(* CODESYS project library.library
   Company: SLAC
   Title: lcls-twincat-motion
   Placeholder: lcls-twincat-motion
   Version: 0.2.0

Project tree, tasks and I/O mapping:
  libraries: Tc2_EtherCAT, * (Beckhoff Automation GmbH); Tc2_MC2, * (Beckhoff Automation GmbH); Tc2_Standard, * (Beckhoff Automation GmbH); Tc2_System, * (Beckhoff Automation GmbH); Tc2_Utilities, * (Beckhoff Automation GmbH); Tc3_Module, * (Beckhoff Automation GmbH); TcUnit, * (www.tcunit.org)
  DUTs/
    data type DUT_MotionStage
    data type DUT_PositionState
    data type EL5042_Status
    data type ENUM_EpicsHomeCmd
    data type ENUM_EpicsMotorCmd
    data type ENUM_StageBrakeMode
    data type ENUM_StageEnableMode
    data type ST_RenishawAbsEnc
  POUs/
    Motion/
      Gantry/
        function block FB_GantryAutoCoupling [ST]
        function block FB_GantryDiffVirtualLimitSwitch [ST]
      function block FB_MotionStage [ST]
      function block FB_SetEnables [ST]
      function block FB_StatePTPMove [ST]
    MotorTesting/
      function block FB_MicroStepCountTest [ST]
  tc_mca_std_lib/
    DUTs/
      data type DUT_AxisStatus_v0_01
    GVLs/
      global variables GVL
    POUs/
      ChangeConfig/
        function block FB_ReadFloatParameter [ST]
        function block FB_ReadParameterInNc_v1_00 [ST]
        function block FB_WriteFloatParameter [ST]
        function block FB_WriteParameterInNc_v1_00 [ST]
      ErrorHandling/
        data type DUT_ErrorState
        data type DUT_TerminalError
        function block FB_ErrorList [ST]
        function block FB_TerminalError [ST]
        global variables GVL_ErrorSystem
        data type ST_ErrorSystem
      Hardware/
        EtherCAT_Terminals/
          Analog_Inputs/
            function block EL3174_0002 [ST]
            function block EL3214 [ST]
            function block EL3255 [ST]
            function block FB_CalculateFrequency_3702_v0_01 [ST]
          Digital_Inputs/
            function block EL1008 [ST]
            function block EL1018 [ST]
            function block EL1808 [ST]
            function block EL1809 [ST]
            function block EL1819 [ST]
            function block FB_EL1252ASM_v1_00 [ST]
          Digital_Outputs/
            External_Types/
              data type dutEL2521_Ctrl
              data type dutEL2521_Status
            function block EL2014 [ST]
            function block EL2252 [ST]
            function block EL2808 [ST]
            function block EL2819 [ST]
          Measuring_Terminals/
            function block EL5002 [ST]
            function block EL5021 [ST]
            function block EL5042 [ST]
            function block EL5101 [ST]
          Motion/
            function block EL7211_v1_00 [ST]
            function block EL9576_v1_00 [ST]
          System/
            function block EL9410 [ST]
            function block EL9505 [ST]
        Other/
          function block EK1200 [ST]
      Motion/
        Homing/
          function block FB_HomeDirect [ST]
          function block FB_HomeFinish [ST]
          function block FB_HomePrepare [ST]
          function block FB_HomeReadNcVelocities [ST]
          function block FB_HomeReadSoftLimEnable [ST]
          function block FB_HomeToSwitch [ST]
          function block FB_HomeVirtual [ST]
          function block FB_HomeWriteNcVelocities [ST]
          function block FB_HomeWriteSoftLimEnable [ST]
        function block FB_DriveVirtual [ST]
        function block FB_NcAxis [ST]
  UnitTests/
    program Interactive [ST]
  Version/
    global variables Global_Version
*)

// DUTs/DUT_MotionStage
TYPE DUT_MotionStage :
STRUCT
	// Hardware
	Axis: AXIS_REF;
	bLimitForwardEnable AT %I*: BOOL;
	bLimitBackwardEnable AT %I*: BOOL;
	bHome AT %I*: BOOL;

	bBrakeRelease AT %Q*: BOOL;
	
	// Psuedo-hardware
	bAllForwardEnable: BOOL:=FALSE; // Forward enable EPS summary
	bAllBackwardEnable: BOOL:=FALSE; // Forward enable EPS summary
	bHardwareEnable AT %I*: BOOL; // True when Emergency stop button is not activated
	
	bAllEnable: BOOL:=FALSE; // Enable EPS summary encapsulating emergency stop button and any additional motion preventive hardware

	bGantryForwardEnable: BOOL:=FALSE; // Forward virtual gantry limit switch
	bGantryBackwardEnable: BOOL:=FALSE; // Reverse virtual gantry limit switch
	
	// Settings
	bPowerSelf: BOOL:=TRUE;
	nEnableMode: INT:=ENUM_StageEnableMode.STAGE_ENABLE_MOTION;
	nBrakeMode: INT:=ENUM_StageBrakeMode.STAGE_BRAKE_DISABLED;
	nHomingMode: INT:=ENUM_EpicsHomeCmd.EPICS_MOTOR_HOME_NONE;
	
	bGantryAxis: BOOL:=FALSE; // Set true to activate gantry EPS
	nGantryTol: LINT:=0; // Set to gantry difference tolerance
	nEncRef: ULINT:=0; // Encoder count at which this axis is aligned with other axis
	
	// Commands
	bEnable: BOOL;
	bReset: BOOL;
	bExecute: BOOL;
	
	// Args
	nCommand: INT;
	nCmdData: INT;
	fPosition: LREAL;
	fVelocity: LREAL;
	fAcceleration: LREAL;
	fDeceleration: LREAL;
	fHomePosition: LREAL;
	
	// Info
	nMotionAxisID: UDINT:=0;
	
	// Returns
	bEnableDone: BOOL;
	bBusy: BOOL;
	bDone: BOOL;
	bError: BOOL;
	sErrorMessage: STRING;
	stAxisStatus: DUT_AxisStatus_v0_01;
END_STRUCT
END_TYPE

// DUTs/DUT_PositionState
TYPE DUT_PositionState :
// Include io: input on things that should never be mutable in EPICS.
// Omit io on things that may or may not need to be mutable, allow engineer to decide in their pragma.
// Currently: some installations would want position and delta to be mutable.
STRUCT
	{attribute 'pytmc' := '
		pv: NAME
		io: input
	'}
	sName: STRING;

	{attribute 'pytmc' := '
		pv: SETPOINT
	'}
	fPosition: LREAL;
	
	{attribute 'pytmc' := '
		pv: DELTA
	'}
	fDelta: LREAL;
	
	{attribute 'pytmc' := '
		pv: VELO
		io: input
	'}
	fVelocity: LREAL;
	
	{attribute 'pytmc' := '
		pv: ACCL
		io: input
	'}
	fAccel: LREAL;
	
	{attribute 'pytmc' := '
		pv: DCCL
		io: input
	'}
	fDecel: LREAL;
END_STRUCT
END_TYPE

// DUTs/EL5042_Status
TYPE EL5042_Status :
STRUCT
END_STRUCT
END_TYPE

// DUTs/ENUM_EpicsHomeCmd
{attribute 'qualified_only'}
{attribute 'strict'}
TYPE ENUM_EpicsHomeCmd :
(
	EPICS_MOTOR_HOME_LLS := 1, // Low limit switch
	EPICS_MOTOR_HOME_HLS := 2, // High limit switch
	EPICS_MOTOR_HOME_LHS := 3, // Home switch via low switch
	EPICS_MOTOR_HOME_HHS := 4, // Home switch via high switch
	EPICS_MOTOR_HOME_ABS := 15, // Set here to be fHomePosition
	EPICS_MOTOR_HOME_NONE := -1 // Do not home, ever
);
END_TYPE

// DUTs/ENUM_EpicsMotorCmd
{attribute 'qualified_only'}
{attribute 'strict'}
TYPE ENUM_EpicsMotorCmd :
(
	EPICS_MOTOR_JOG := 0,
	EPICS_MOTOR_MOVE_VEL := 1,
	EPICS_MOTOR_MOVE_REL := 2,
	EPICS_MOTOR_MOVE_ABS := 3,
	EPICS_MOTOR_MOVE_MOD := 4,
	EPICS_MOTOR_HOME := 10,
	EPICS_MOTOR_GEAR := 30
);
END_TYPE

// DUTs/ENUM_StageBrakeMode
{attribute 'qualified_only'}
{attribute 'strict'}
TYPE ENUM_StageBrakeMode :
(
	STAGE_BRAKE_DISABLED,
	STAGE_BRAKE_STANDSTILL
);
END_TYPE

// DUTs/ENUM_StageEnableMode
{attribute 'qualified_only'}
{attribute 'strict'}
TYPE ENUM_StageEnableMode :
(
	STAGE_ENABLE_ALWAYS, // Always set bEnable to TRUE
	STAGE_ENABLE_NEVER,  // Only change bEnable on errors
	STAGE_ENABLE_MOTION  // Enable before motion, disable after motion
);
END_TYPE

// DUTs/ST_RenishawAbsEnc
// Renishaw BiSS-C absolute encoder used with an EL5042 
TYPE ST_RenishawAbsEnc :
STRUCT
	Count AT %I*: ULINT; // Connect to encoder "Position" input
	Status: EL5042_Status; // Status struct placeholder
	Ref: ULINT; // Encoder zero position (useful for aligned position with gantries)
END_STRUCT
END_TYPE

// tc_mca_std_lib/DUTs/DUT_AxisStatus_v0_01
TYPE DUT_AxisStatus_v0_01 :
STRUCT
	bEnable: BOOL;
	bReset: BOOL;
	bExecute: BOOL;
	nCommand: UINT;
	nCmdData: UINT;
	fVelocity: LREAL;
	fPosition: LREAL;
	fAcceleration: LREAL;
	fDeceleration: LREAL;
	bJogFwd: BOOL;
	bJogBwd: BOOL;
	bLimitFwd: BOOL;
	bLimitBwd: BOOL;
	fOverride: LREAL := 100;
	bHomeSensor: BOOL;
	bEnabled: BOOL;
	bError: BOOL;
	nErrorId: UDINT;
	fActVelocity: LREAL;
	fActPosition: LREAL;
	fActDiff: LREAL;
	bHomed:BOOL;
	bBusy:BOOL;
END_STRUCT
END_TYPE

// tc_mca_std_lib/POUs/ErrorHandling/DUT_ErrorState
{attribute 'qualified_only'}
{attribute 'strict'}
TYPE DUT_ErrorState :
(
	None,
	Active,
	Inactive,
	Acknowledged
);
END_TYPE

// tc_mca_std_lib/POUs/ErrorHandling/DUT_TerminalError
TYPE DUT_TerminalError :
STRUCT
	//Error system related
	iTerminalID : INT;					//ID of the terminal
	Error_ID : ULINT := 0;				//ID for the Error entry
	ErrorState : DUT_ErrorState;		//State of the error
	
	//Error related
	nDateTimeOn : ULINT;				//Date and time when the error occured. Raw data
	sDateTimeOn : STRING(24);			//Date and time when the error occured. Readable format
	nDateTimeOff : ULINT;				//Date and time when the error disapeared. Raw data
	sDateTimeOff : STRING(24);			//Date and time when the error disapeared. Readable format
	bWcState : BOOL;					//WcState variable of the terminal
	uiInfoDataState : UINT;				//InfoData.State variable of the terminal
	sErrorMessage : STRING (128);		//Error message corresponding to WcState and InfoData.State
	ErrorType : INT; 					//Error types (priorities) need to be developed
END_STRUCT
END_TYPE

// tc_mca_std_lib/POUs/ErrorHandling/ST_ErrorSystem
TYPE ST_ErrorSystem :
STRUCT
	//Array of error data. Size = cSizeOfErrorData in the GVL
	aErrorData : ARRAY [0..GVL_ErrorSystem.cSizeOfErrorData - 1] OF DUT_TerminalError;
	lNextErrorID : ULINT := 1;					//ErrorID for the next error entry
	nNoErrors : UINT;							//Number of errors in the list
	nNoOverflows : INT := 0;					//Number of overflows. How many error entries have been lost
END_STRUCT
END_TYPE

// tc_mca_std_lib/POUs/Hardware/EtherCAT_Terminals/Digital_Outputs/External_Types/dutEL2521_Ctrl
TYPE dutEL2521_Ctrl :
STRUCT
	///The control word (CW) is located in the output process image, and is transmitted from the controller to the terminal.
	///CW.0 FREQ_SEL 0bin / 1bin  Rapid change of the base frequency (only if the ramp function is inactive):
	///0bin = Base frequency 1 (object 8001:02)
	///1bin = Base frequency 2 (object 8001:03) 
	FREQ_SEL: BOOL;
	///CW.1 RAMP_DIS 1bin Operation of the ramp function is cancelled, in spite of object 8000:06 being active; if travel distance control is active, it is interrupted by this bit 
	RAMP_DIS: BOOL;
	///CW.2 GO_COUNTER 1bin  If travel distance control is active (object 8000:0A), then a pre-set counter value is approached when the bit is set 
	GO_COUNTER: BOOL;
	///CW.5 CNT_CLR 1bin The contents of the counter is cleared or set (object 8000:0B) by this bit. 
	///Any overflow or underflow bits that might be set are also cleared by this bit. 
	///The process can be edge triggered or level triggered (object 8000:05). 
	CNT_CLR: BOOL;
END_STRUCT
END_TYPE

// tc_mca_std_lib/POUs/Hardware/EtherCAT_Terminals/Digital_Outputs/External_Types/dutEL2521_Status
TYPE dutEL2521_Status :
STRUCT
	///The status word (SW) is located in the input process image, and is transmitted from the terminal to the controller.
	///SW.0 SEL_ACK/END_COUNTER 1bin  Confirms the change of base frequency. At activated travel distance control: target counter value reached 
	SEL_ACK: BOOL;
	///SW.1 RAMP_ACTIVE 1bin Ramp is currently being followed 
	RAMP_ACTIVE: BOOL;
	///SW.2 UNDERFLOW 1bin This bit is set if the 16-bit counter underflows (0 -> 65535). It is reset when the counter drops below two thirds of its measuring range (43690 -> 43689) or immediately an overflow occurs. 
	UNDERFLOW: BOOL;
	///SW.3 OVERFLOW 1bin This bit is set if the 16-bit counter overflows (65535 -> 0). It is reset when the counter exceeds one third of its measuring range (21845 -> 21846) or immediately an underflow occurs 
	OVERFLOW: BOOL;
	///SW.4 INPUT_T 1bin Status of INPUT_T 
	INPUT_T: BOOL;
	///SW.5 INPUT_Z 1bin Status of INPUT_Z 
	INPUT_Z: BOOL;
	///SW.6 ERROR 1bin General error bit, included with overflow/underflow 
	ERROR: BOOL;
END_STRUCT
END_TYPE

// tc_mca_std_lib/GVLs/GVL
VAR_GLOBAL
	nHomingError:UDINT:=16#14D00;
END_VAR

// tc_mca_std_lib/POUs/ErrorHandling/GVL_ErrorSystem
{attribute 'qualified_only'}
VAR_GLOBAL CONSTANT
	cSizeOfErrorData : UINT := 128;
	
END_VAR

// Version/Global_Version
{attribute 'TcGenerated'}
// This function has been automatically generated from the project information.
VAR_GLOBAL CONSTANT
	{attribute 'const_non_replaced'}
	{attribute 'linkalways'
	stLibVersion_lcls-twincat-motion : ST_LibVersion := (iMajor := 0, iMinor := 2, iBuild := 0, iRevision := 0, sVersion := '0.2.0');
END_VAR

// POUs/Motion/Gantry/FB_GantryAutoCoupling
FUNCTION_BLOCK FB_GantryAutoCoupling
VAR_INPUT
	nGantryTol : LINT;
END_VAR
VAR_OUTPUT
	bGantryAlreadyCoupled : BOOL;
END_VAR
VAR_IN_OUT
	Master : DUT_MotionStage;
	MasterEnc : ST_RenishawAbsEnc;
	Slave : DUT_MotionStage;
	SlaveEnc : ST_RenishawAbsEnc;
	bExecuteCouple : BOOL;
	bExecuteDecouple : BOOL;
END_VAR
VAR
	gantry_diff_limit : FB_GantryDiffVirtualLimitSwitch;
	couple : MC_GEARIN;
	decouple : MC_GEAROUT;
	bInitComplete : BOOL;
	fbSetEnables : FB_SetEnables;
END_VAR

// Designate Master and SLave Axes
Master.bGantryAxis := TRUE;
Slave.bGantryAxis := TRUE;

Master.nGantryTol := nGantryTol;
Slave.nGantryTol := Master.nGantryTol;

// Activate Gantry Virtual Limit Switch
gantry_diff_limit(Penc:=MasterEnc, SEnc:=SlaveEnc, GantDiffTol:=Master.nGantryTol,
				  PLimFwd=>Master.bGantryForwardEnable, PLimBwd=>Master.bGantryBackwardEnable,
				  SLimFwd=>Slave.bGantryForwardEnable, SLimBwd=>Slave.bGantryBackwardEnable);

// Coupling Status Bit
bGantryAlreadyCoupled := Master.Axis.NcToPlc.CoupleState=1 AND Slave.Axis.NcToPlc.CoupleState=3;

fbSetEnables(stMotionStage:=Master);
fbSetEnables(stMotionStage:=Slave);

IF bGantryAlreadyCoupled THEN
	Master.bGantryForwardEnable := Master.bGantryForwardEnable AND Slave.bAllForwardEnable;
	Slave.bGantryForwardEnable := Master.bAllForwardEnable AND Slave.bGantryForwardEnable;
	
	Master.bGantryBackwardEnable := Master.bGantryBackwardEnable AND Slave.bAllBackwardEnable;
	Slave.bGantryBackwardEnable := Master.bAllBackwardEnable AND Slave.bGantryBackwardEnable;
END_IF


// Coupling states
// Auto-coupling at init and auto-reset of coupling boolean
bExecuteCouple S= NOT bInitComplete;

bExecuteCouple R= couple.Busy OR bGantryAlreadyCoupled;
couple(Master:=Master.Axis, Slave:=Slave.Axis, Execute:=bExecuteCouple);

bInitComplete S= bGantryAlreadyCoupled;

// Decoupling with auto-reset of coupling boolean
bExecuteDecouple R= decouple.Busy OR NOT bGantryAlreadyCoupled;
decouple(Slave:=Slave.Axis, Execute:=bExecuteDecouple);

END_FUNCTION_BLOCK

// POUs/Motion/Gantry/FB_GantryDiffVirtualLimitSwitch
FUNCTION_BLOCK FB_GantryDiffVirtualLimitSwitch
VAR_INPUT
	PEnc: ST_RenishawAbsEnc; // Primary axis encoder (usually the upstream one)
	SEnc: ST_RenishawAbsEnc; // Secondary axis encoder (couples to the primary)
	
	GantDiffTol: LINT;		// Gantry differenace tolerance in encoder counts
END_VAR
VAR_OUTPUT
	PLimFwd: BOOL; // Primary axis forward direction enable
	PLimBwd: BOOL; // Primary axis reverse direction enable
	SLimFwd: BOOL; // Secondary axis forward direction enable
	SLimBwd: BOOL; // Secondary axis reverse direction enable
END_VAR
VAR
	GantryDiff: LINT;
END_VAR

(* Gantry Difference Virtual Limit Switch
A. Wallace 2017-2-15

Determines which direction is disabled due to it increasing the gantry difference.
Refer to the ESD for actual conventions.

A positive gantry error refers to a CCW clocked assembly:
eg. for X
X1 upstream, X2 downstream. Primary axis is always upstream.
Gantry difference > 0 when
X2>X1
Therefore
X2 positive direction disabled
X1 negative direction disabled

Call before FB_MotionStage fb calls for the gantry axes.
*)

GantryDiff := ( ULINT_TO_LINT(PEnc.Count) - ULINT_TO_LINT(PEnc.Ref) ) - ( ULINT_TO_LINT(SEnc.Count) - ULINT_TO_LINT(SEnc.Ref) );

IF ABS(GantryDiff) > GantDiffTol THEN
	IF GantryDiff < 0  THEN
		PLimBwd := FALSE;
		SLimFwd := FALSE;
	ELSE	
		PLimBwd := TRUE;
		SLimFwd := TRUE;
	END_IF
	IF GantryDiff > 0 THEN
		PLimFwd := FALSE;
		SLimBwd := FALSE;
	ELSE
		PLimFwd := TRUE;
		SLimBwd := TRUE;
	END_IF
ELSE
	//If there is no fault, all directions are enabled
	PLimFwd := TRUE;
	PLimBwd := TRUE;
	SLimFwd := TRUE;
	SLimBwd := TRUE;
END_IF

END_FUNCTION_BLOCK

// POUs/Motion/FB_MotionStage
FUNCTION_BLOCK FB_MotionStage
VAR_IN_OUT
	stMotionStage: DUT_MotionStage;
END_VAR
VAR
	fbDriveVirtual: FB_DriveVirtual;
	bExecute: BOOL;
	bFwdHit: BOOL;
	bBwdHit: BOOL;
	fbExecFallingEdge: F_TRIG;
	fbSetEnables: FB_SetEnables;
END_VAR

// Start with an accurate status
stMotionStage.Axis.ReadStatus();

// Handle auto-enable timing
CASE stMotionStage.nEnableMode OF
	ENUM_StageEnableMode.STAGE_ENABLE_ALWAYS:
		stMotionStage.bEnable := TRUE;
		bExecute := stMotionStage.bExecute;
	ENUM_StageEnableMode.STAGE_ENABLE_NEVER:
		bExecute := stMotionStage.bExecute;
	ENUM_StageEnableMode.STAGE_ENABLE_MOTION:
		IF stMotionStage.bExecute THEN
			stMotionStage.bEnable := TRUE;
		END_IF
		bExecute := stMotionStage.bExecute AND stMotionStage.bEnableDone;
END_CASE

// Automatically fill the correct nCmdData for homing
IF stMotionStage.nCommand = ENUM_EpicsMotorCmd.EPICS_MOTOR_HOME THEN
	stMotionStage.nCmdData := stMotionStage.nHomingMode;
END_IF

fbSetEnables(stMotionStage:=stMotionStage);

// Handle standard commands using ESS's FB
fbDriveVirtual(En:=TRUE,
	bEnable:=stMotionStage.bAllEnable,
	bReset:=stMotionStage.bReset,
	bExecute:=bExecute,
	nCommand:=INT_TO_UINT(stMotionStage.nCommand),
	nCmdData:=INT_TO_UINT(stMotionStage.nCmdData),
	fVelocity:=stMotionStage.fVelocity,
	fPosition:=stMotionStage.fPosition,
	fAcceleration:=stMotionStage.fAcceleration,
	fDeceleration:=stMotionStage.fDeceleration,
	bLimitFwd:=stMotionStage.bAllForwardEnable,
	bLimitBwd:=stMotionStage.bAllBackwardEnable,
	bHomeSensor:=stMotionStage.bHome,
	fHomePosition:=stMotionStage.fHomePosition,
	bPowerSelf:=stMotionStage.bPowerSelf,
	nMotionAxisID=>stMotionStage.nMotionAxisID,
	bError=>stMotionStage.bError,
	sErrorMessage=>stMotionStage.sErrorMessage,
	Axis:=stMotionStage.Axis);

IF fbDriveVirtual.bBusy THEN
	stMotionStage.bBusy := TRUE;
	stMotionStage.bDone := FALSE;
END_IF

IF stMotionStage.bError THEN
	stMotionStage.bBusy := FALSE;
	stMotionStage.bDone := FALSE;
	stMotionStage.bEnable := FALSE;
END_IF

// Check the limits and cancel execution if appropriate. Without this block we have infinite error spam
bFwdHit := stMotionStage.Axis.Status.PositiveDirection AND NOT stMotionStage.bAllForwardEnable;
bBwdHit := stMotionStage.Axis.Status.NegativeDirection AND NOT stMotionStage.bAllBackwardEnable;
IF bFwdHit OR bBwdHit THEN
	stMotionStage.bExecute := FALSE;
END_IF

// Mark done if settled or if unexpected stop, then reset the FB if there is no error
fbExecFallingEdge(CLK:=stMotionStage.bExecute);
IF (stMotionStage.Axis.Status.InTargetPosition AND NOT fbDriveVirtual.bBusy) OR fbExecFallingEdge.Q THEN
	IF NOT stMotionStage.bDone THEN
		stMotionStage.bDone := TRUE;
		stMotionStage.bBusy := FALSE;
		IF NOT stMotionStage.Axis.Status.Error THEN
			bExecute := FALSE;
			stMotionStage.bExecute := FALSE;
		END_IF
	END_IF
END_IF
IF stMotionStage.nEnableMode = ENUM_StageEnableMode.STAGE_ENABLE_MOTION AND NOT bExecute THEN
	IF stMotionStage.Axis.Status.MotionState = MC_AXISSTATE_STANDSTILL THEN
		stMotionStage.bEnable := FALSE;
	END_IF
END_IF

// Get a definitive bEnabled reading
CASE stMotionStage.Axis.Status.MotionState OF
	// We are not enabled if there is an issue
	MC_AXISSTATE_UNDEFINED, MC_AXISSTATE_DISABLED, MC_AXISSTATE_ERRORSTOP:
		stMotionStage.bEnableDone := FALSE;
	ELSE
		stMotionStage.bEnableDone := TRUE;
END_CASE

// Handle the brake. TRUE means brake disabled.
CASE stMotionStage.nBrakeMode OF
	ENUM_StageBrakeMode.STAGE_BRAKE_DISABLED:
		stMotionStage.bBrakeRelease := stMotionStage.bEnableDone AND stMotionStage.bExecute;
	ENUM_StageBrakeMode.STAGE_BRAKE_STANDSTILL:
		IF stMotionStage.Axis.Status.MotionState = MC_AXISSTATE_STANDSTILL THEN
			stMotionStage.bBrakeRelease := FALSE;
		ELSE
			stMotionStage.bBrakeRelease := TRUE;
		END_IF
END_CASE
CASE stMotionStage.Axis.Status.MotionState OF
	MC_AXISSTATE_UNDEFINED, MC_AXISSTATE_ERRORSTOP:
		stMotionStage.bBrakeRelease := FALSE;
END_CASE

// Sync the epics status struct
stMotionStage.stAxisStatus := fbDriveVirtual.stAxisStatus;
stMotionStage.stAxisStatus.bEnabled := stMotionStage.bEnableDone;

// Reset everything when bReset is flagged
IF stMotionStage.bReset THEN
	stMotionStage.bEnable := FALSE;
	stMotionStage.bReset := FALSE;
	stMotionStage.bExecute := FALSE;
	bExecute := FALSE;
END_IF

// Ignore homing if we have the setting for it
// e.g. for pre-calibrated absolute encoders
IF stMotionStage.nHomingMode = ENUM_EpicsHomeCmd.EPICS_MOTOR_HOME_NONE THEN
	stMotionStage.stAxisStatus.bHomed := TRUE;
END_IF

END_FUNCTION_BLOCK

// tc_mca_std_lib/POUs/Motion/FB_DriveVirtual
///#########################################################
///Function block to run a virtual drive with Nc
///	Library:		
///	Tc2_MC2.lib
///
///	Global Variables:
///	
///	Data types:
///	
///	External functions:
///
///###########################################################
FUNCTION_BLOCK FB_DriveVirtual
VAR
	sVersion: STRING:='1.0.3';	
END_VAR
VAR_INPUT
	En: BOOL;
	bEnable: BOOL;
	bReset: BOOL;
	bExecute: BOOL;
	/////	nCommandLocal...
	/////	0 = Jog
	/////	1 = MoveVelocity
	/////	2 = MoveRelative
	/////	3 = MoveAbsolut
	/////	4 = MoveModulo
	/////	10 = Homing
	/////	20 = SuperInp >>>ToBe
	/////	30 = Gear
	nCommand: UINT;
	nCmdData: UINT;
	fVelocity: LREAL;
	fPosition: LREAL;
	fAcceleration: LREAL;
	fDeceleration: LREAL;
	bJogFwd: BOOL;
	bJogBwd: BOOL;
	bLimitFwd: BOOL;
	bLimitBwd: BOOL;	
	fOverride: LREAL := 100;
	bHomeSensor: BOOL;
	fHomePosition:LREAL;
	nHomeRevOffset: UINT;
	MasterAxis: AXIS_REF;
	bPowerSelf: BOOL;
END_VAR
VAR_OUTPUT
	EnO: BOOL;
	bEnabled: BOOL;
	bBusy: BOOL;
	bDone: BOOL;
	bError: BOOL;
	bHomed: BOOL;
	nErrorId: UDINT;
	nMotionAxisID:UDINT:=0;  //Axis id in Motion (NC)
	Status: ST_AxisStatus;
	fActVelocity: LREAL;
	fActPosition: LREAL;
	fActDiff: LREAL;
    sErrorMessage:STRING;
END_VAR
VAR_IN_OUT
	Axis: AXIS_REF;
END_VAR
VAR	
	nCommandLocal: UINT;
	nCmdDataLocal: UINT;
	bFirstScan: BOOL := TRUE;
	fbReset: MC_Reset;
	fbPower: MC_Power;
	fbHalt: MC_Halt;
	fbJog: MC_Jog;
	fbMoveVelocity: MC_MoveVelocity;
	fbMoveRelative: MC_MoveRelative;
	fbMoveAbsolute: MC_MoveAbsolute;
	fbMoveModulo: MC_MoveModulo;	
	fbHomeVirtual:FB_HomeVirtual;
	fbGearInDyn: MC_GearInDyn;
	fbGearOut: MC_GearOut;
	fbExecuteRiseEdge: R_TRIG;
	stAxisStatus: DUT_AxisStatus_v0_01;	
END_VAR

EnO:=En;

// Transfer nCommand and nCmdData to local copies at rising edge of bExecute (avoid issues if nCommand or nCmdData are changed during a command) 
fbExecuteRiseEdge(CLK:=bExecute);
IF fbExecuteRiseEdge.Q THEN
  nCmdDataLocal:=nCmdData;
  nCommandLocal:=nCommand;
END_IF

bHomed:=fbHomeVirtual.bHomed; //Add in DUT_AxisStatus later
bDone:=FALSE;

(*Reset*)
fbReset(
	Execute:=bReset AND Axis.Status.Error,
	Axis:=Axis,
	Done=> ,
	Busy=> ,
	Error=> ,
	ErrorID=> );

(*Power*)
IF bPowerSelf THEN
fbPower(
	Axis:=Axis,
	Enable:=bEnable,	
	Enable_Positive:=bEnable AND bLimitFwd,	
	Enable_Negative:=bEnable AND bLimitBwd,	
	Override:=fOverride,
	BufferMode:= ,
	Status=> ,
	Busy=> ,
	Active=> ,
	Error=> ,
	ErrorID=> );
END_IF

(*Halt*)
fbHalt(
	Execute:=NOT bExecute  AND (((fbMoveVelocity.Busy OR fbPower.Busy) AND (nCommandLocal=1)) OR (fbMoveRelative.Busy AND (nCommandLocal=2)) OR (fbMoveAbsolute.Busy AND (nCommandLocal=3)) OR (fbMoveModulo.Busy AND (nCommandLocal=4)) OR (fbHomeVirtual.bBusy AND (nCommandLocal=10))),
	Deceleration:=fDeceleration,
	Jerk:=0,
	BufferMode:= ,
	Options:= ,
	Axis:=Axis ,
	Done=> ,
	Busy=> ,
	Active=> ,
	CommandAborted=> ,
	Error=> ,
	ErrorID=> );

(*Jog (Command = 0)*)
fbJog(
	JogForward:=bJogFwd AND (nCommandLocal=0) ,
	JogBackwards:=bJogBwd AND (nCommandLocal=0) ,
	Mode:=UINT_TO_INT(nCmdDataLocal),
	Position:= ,
	Velocity:=fVelocity,
	Acceleration:=fAcceleration,
	Deceleration:=fDeceleration,
	Jerk:=0,
	Axis:=Axis,
	Done=> ,
	Busy=> ,
	Active=> ,
	CommandAborted=> ,
	Error=> ,
	ErrorID=> );

(*MoveVelocity (Command = 1)*)
fbMoveVelocity(
	Execute:=bExecute AND (nCommandLocal=1),
	Velocity:=ABS(fVelocity),
	Acceleration:=fAcceleration,
	Deceleration:=fDeceleration,
	Jerk:=0,
	Direction:=SEL(fVelocity<0, MC_Positive_Direction, MC_Negative_Direction),
	BufferMode:= ,
	Options:= ,
	Axis:=Axis,
	InVelocity=> ,
	Busy=> ,
	Active=> ,
	CommandAborted=> ,
	Error=> ,
	ErrorID=> );

(*MoveRelative (Command = 2)*)
fbMoveRelative(
	Execute:=bExecute AND (nCommandLocal=2), 
	Distance:=fPosition, 
	Velocity:=ABS(fVelocity), 
	Acceleration:=fAcceleration,
	Deceleration:=fDeceleration,
	Jerk:=0,
	BufferMode:= , 
	Options:= , 
	Axis:=Axis, 
	Done=> , 
	Busy=> , 
	Active=> , 
	CommandAborted=> , 
	Error=> , 
	ErrorID=> );
	
IF nCommandLocal=2 THEN
	bDone:=fbMoveRelative.Done;
END_IF
	
(*MoveAbsolute (Command = 3)*)
fbMoveAbsolute(
	Execute:=bExecute AND (nCommandLocal=3),
	Position:=fPosition,
	Velocity:=ABS(fVelocity),
	Acceleration:=fAcceleration,
	Deceleration:=fDeceleration,
	Jerk:=0,
	BufferMode:= ,
	Options:= ,
	Axis:=Axis,
	Done=> ,
	Busy=> ,
	Active=> ,
	CommandAborted=> ,
	Error=> ,
	ErrorID=> );

IF nCommandLocal=3 THEN
	bDone:=fbMoveAbsolute.Done;
END_IF

(*MoveModulo (Command = 4)*)
fbMoveModulo(
	Execute:=bExecute AND (nCommandLocal=4), 
	Position:=fPosition, 
	Velocity:=ABS(fVelocity), 
	Acceleration:=fAcceleration, 
	Deceleration:=fDeceleration, 
	Jerk:=0, 
	Direction:=UINT_TO_INT(nCmdDataLocal), 
	BufferMode:= , 
	Options:= , 
	Axis:=Axis, 
	Done=> , 
	Busy=> , 
	Active=> , 
	CommandAborted=> , 
	Error=> , 
	ErrorID=> );

IF nCommandLocal=4 THEN
	bDone:=fbMoveModulo.Done;
END_IF
	
(*Home (Command = 10)*)
fbHomeVirtual(	
	bExecute:= nCommandLocal=10 AND bExecute,
	fHomePosition:=fHomePosition,
	bHomeSensor:=bHomeSensor,
	bLimitBwd:=bLimitBwd,
	bLimitFwd:=bLimitFwd,
	nCmdData:=nCmdDataLocal,
	bReset:=bReset,
	nHomeRevOffset:=nHomeRevOffset,
	Axis:=Axis
	);
	
IF nCommandLocal=10 THEN
	bDone:=fbHomeVirtual.bDone;
END_IF
	
(*Gear (Command = 30)*)
fbGearInDyn(
	Enable:=bExecute  AND (nCommandLocal=30),
	GearRatio:=SEL(nCmdDataLocal>0, 1,fVelocity),
	Acceleration:=fAcceleration,
	Deceleration:=fDeceleration,
	Jerk:=0.0,
	BufferMode:= , 
	Options:= , 
	Master:=MasterAxis,
	Slave:=Axis,
	InGear=> , 
	Busy=> , 
	Active=> , 
	CommandAborted=> , 
	Error=> , 
	ErrorID=> );
	
fbGearOut(
	Execute:=NOT bExecute AND Axis.Status.NotMoving AND (nCommandLocal=30),
	Slave:=Axis,
	Error=>,
	Done=>,
	ErrorID=>);


IF nCommandLocal=30 THEN
	bDone:=Axis.Status.Coupled;
END_IF

(*Busy*)
bBusy:=Axis.Status.HasJob OR Axis.Status.HomingBusy OR fbHomeVirtual.bBusy;

(*Enabled*)
bEnabled:=fbPower.Status;

(*Error from functions and Nc*)
IF fbPower.Error AND fbPower.Active THEN
	bError:=fbPower.Enable;
	nErrorId:=fbPower.ErrorID;
ELSIF fbHalt.Error AND fbHalt.Active THEN
	bError:=fbHalt.Execute;
	nErrorId:=fbHalt.ErrorID;
ELSIF fbJog.Error AND nCommandLocal=0 (*fbJog.Active*) THEN
	bError:=fbJog.JogForward OR fbJog.JogBackwards;
	nErrorId:=fbJog.ErrorID;
ELSIF fbMoveVelocity.Error AND nCommandLocal=1(*fbMoveVelocity.Active*) THEN
	bError:=fbMoveVelocity.Execute;
	nErrorId:=fbMoveVelocity.ErrorID;
ELSIF fbMoveRelative.Error AND nCommandLocal=2 (*fbMoveRelative.Active*) THEN
	bError:=fbMoveRelative.Execute;
	nErrorId:=fbMoveRelative.ErrorID;
ELSIF fbMoveAbsolute.Error AND nCommandLocal=3 (*fbMoveAbsolute.Active*) THEN
	bError:=fbMoveAbsolute.Execute;
	nErrorId:=fbMoveAbsolute.ErrorID;
ELSIF fbMoveModulo.Error AND nCommandLocal=4 (*fbMoveModulo.Active*) THEN
	bError:=fbMoveModulo.Execute;
	nErrorId:=fbMoveModulo.ErrorID;
ELSIF fbHomeVirtual.bError AND nCommandLocal=10 (*fbHome.Active*) THEN
	bError:=fbHomeVirtual.bError;
	nErrorId:=fbHomeVirtual.nErrorID;
ELSIF fbGearInDyn.Error AND nCommandLocal=30 (*fbGearInDyn.Active*) THEN
	bError:=fbGearInDyn.Enable;
	nErrorId:=fbGearInDyn.ErrorID;
ELSIF fbGearOut.Error AND nCommandLocal=30 AND Axis.Status.Coupled THEN
	bError:=fbGearOut.Execute;
	nErrorId:=fbGearOut.ErrorID;
ELSIF Axis.Status.Error  THEN
	bError:=TRUE;
	nErrorId:=Axis.Status.ErrorID;
ELSIF fbHomeVirtual.bError THEN
	bError:=TRUE;
	nErrorId:=fbHomeVirtual.nErrorId;
ELSE
	bError:=FALSE;
	nErrorId:=0;
END_IF;

(*Converese nErrorID to string*)
sErrorMessage:=WORD_TO_HEXSTR(in:=TO_WORD(nErrorID) , iPrecision:= 4, bLoCase:=0 );

(*Status from Nc*)
Status:=Axis.Status;

(*Axis id in motion "motor"*)
nMotionAxisID:=axis.NcToPlc.AxisId;

(*Actual Velocity*)
fActVelocity:=Axis.NcToPlc.ActVelo;

(*Actual Position*)
IF Axis.Status.OpMode.Modulo THEN
	fActPosition:=Axis.NcToPlc.ModuloActPos;
ELSE
	fActPosition:=Axis.NcToPlc.ActPos;
END_IF

(*Actual Position*)
fActDiff:=Axis.NcToPlc.PosDiff;


//Status struct for EPICS communication
stAxisStatus.bEnable:=bEnable;
stAxisStatus.bEnabled:=bEnabled;
stAxisStatus.bError:=bError;
stAxisStatus.bExecute:=bExecute;
stAxisStatus.bHomeSensor:=bHomeSensor;
stAxisStatus.bJogBwd:=bJogBwd;
stAxisStatus.bJogFwd:=bJogFwd;
stAxisStatus.bLimitBwd:=bLimitBwd;
stAxisStatus.bLimitFwd:=bLimitFwd;
stAxisStatus.bReset:=bReset;
stAxisStatus.fAcceleration:=fAcceleration;
stAxisStatus.fActDiff:=fActDiff;
stAxisStatus.fActPosition:=fActPosition;
stAxisStatus.fActVelocity:=fActVelocity;
stAxisStatus.fDeceleration:=fDeceleration;
stAxisStatus.fOverride:=fOverride;
stAxisStatus.fPosition:=fPosition;
stAxisStatus.fVelocity:=fVelocity;
stAxisStatus.nCmdData:=nCmdData;  //Or nCmdDataLocal
stAxisStatus.nCommand:=nCommand;  //Or nCommandLocal
stAxisStatus.nErrorId:=nErrorId;
stAxisStatus.bBusy:=bBusy;
stAxisStatus.bHomed:=bHomed;

IF bFirstScan THEN
	bFirstScan:=FALSE;
END_IF

END_FUNCTION_BLOCK

// tc_mca_std_lib/POUs/Motion/Homing/FB_HomeVirtual
FUNCTION_BLOCK FB_HomeVirtual
VAR_INPUT
	En: BOOL;
	bReset: BOOL;
	bExecute: BOOL;
	nCmdData: UINT;
	bLimitFwd: BOOL;
	bLimitBwd: BOOL;	
	bHomeSensor: BOOL;	
	fHomePosition:LREAL;
	nHomeRevOffset: UINT;
END_VAR
VAR_IN_OUT
	Axis: AXIS_REF;
END_VAR
VAR_OUTPUT
	EnO: BOOL;	
	bBusy: BOOL;
	bDone: BOOL;
	bHomed:BOOL;
	bError: BOOL;
	nErrorId: UDINT;
END_VAR
VAR
	fbHomeToSwitch: FB_HomeToSwitch;
    fbHomeDirect: FB_HomeDirect; //Only used for direct homing (set of position)
    fbMoveVelocity:MC_MoveVelocity;
    fbHomePrepare:FB_HomePrepare;
	fbHomeFinish:FB_HomeFinish;    	    		
	fbExecuteRiseEdge: R_TRIG;
    nHomingState:INT:=0;
	bExecuteHomeToSwitch:BOOL:=FALSE;
	bExecuteMoveVelocity:BOOL:=FALSE;
	bExecutePrepare: BOOL:=FALSE;
	bExecuteFinish: BOOL:=FALSE;
	bExecuteHomeDirect: BOOL;
	nCmdDataLocal: UINT;  //Ensure that nCmdData is not changed during sequence
	bSequenceReady:BOOL:=TRUE;
	bRestoreNCDataNeeded: BOOL:=FALSE;
END_VAR

EnO:=En;

IF bReset THEN	
	bError:=FALSE;
	nErrorId:=0;
END_IF

// Reset when bExecute is low
IF NOT bExecute THEN
  nHomingState:=0;
  bSequenceReady:=TRUE;
  bExecuteHomeToSwitch:=FALSE;
  bExecuteHomeDirect:=FALSE;
  bExecuteMoveVelocity:=FALSE;
  bExecutePrepare:=FALSE;
  bExecuteFinish:=FALSE;
END_IF

//Reset at rinsing edge of bExecute
fbExecuteRiseEdge(CLK:=bExecute);
IF fbExecuteRiseEdge.Q THEN
  nCmdDataLocal:=nCmdData; //Ensure that nCmdData is not changed during sequence (nCmdData will only be read at a rising edge of bExecute)
  bSequenceReady:=FALSE;
  bExecutePrepare:=TRUE;  
  bRestoreNCDataNeeded:=FALSE;
  //Check if valid nCmdDataLocal
  CASE nCmdDataLocal OF  	
    1:
    2:
    3:
    4:
    15:
    ELSE //nCmdData not valid	
      bError:=TRUE;
      nErrorId:=16#4FFF;   
  END_CASE
END_IF

//############# Prepare for homing (Read from NC and reset homed flag)
fbHomePrepare(
  En:=En,
  bExecute:=bExecutePrepare AND NOT bError, // Not needed for sequence 15 (set position only, no movement))
  bReset:=bReset,
  Axis:=Axis,
);

//############# Homing Sequences:
CASE nCmdDataLocal OF  
	
   1: // Home to low limit switch
	   CASE nHomingState OF
		  0:
		    bHomed:=Axis.Status.Homed;
            // Wait for read of velocities from NC and reset of calibration flag
	        IF fbHomePrepare.bDone AND bExecute AND NOT bSequenceReady THEN
			  bRestoreNCDataNeeded:=TRUE;
			  IF bLimitBwd THEN
                nHomingState:=1;
              ELSE
				nHomingState:=2;  //Standing on limit switch go direct to state 2 
              END_IF                                          		  
	        END_IF
		  1: // wait for reach low limit then trigger fbHomeToSwitch
		    bHomed:=FALSE;
			bSequenceReady:=FALSE;
			fbMoveVelocity.Velocity:=ABS(fbHomePrepare.fVelocityToCam);
            fbMoveVelocity.Direction:=MC_Negative_Direction;
	        bExecuteMoveVelocity:=bExecute;  // Execute MC_MoveVelocity
		    IF NOT bLimitBwd AND NOT fbMoveVelocity.Busy AND Axis.Status.NotMoving THEN //MC_MoveVelocity.Busy goes down when ramp down initiates (not ends).
			  nHomingState:=2;
		    END_IF
		  2: // Wait for fbHomeToSwitch
		    bHomed:=FALSE;
		    bSequenceReady:=FALSE;
            bExecuteMoveVelocity:=FALSE;			
            bExecuteHomeToSwitch:=TRUE;	
            fbHomeToSwitch.nSearchDirTwoardsCam:=MC_Positive_Direction;
            fbHomeToSwitch.nSearchDirOffCam:=MC_Positive_Direction;	             
	        fbHomeToSwitch.fVelocityToCamNC:=fbHomePrepare.fVelocityToCam; // High speed
  	        fbHomeToSwitch.fVelocityFromCamNC:=fbHomePrepare.fVelocityFromCam;  // Low speed              		
		    fbHomeToSwitch.bCamSensor:=NOT bLimitBwd;            	 		    
	        IF fbHomeToSwitch.bDone THEN	          
			  nHomingState:=3;
			  bExecuteFinish:=TRUE;
			  fbHomeFinish.bSofLimEnableHigh:=fbHomePrepare.bSofLimEnableHighOriginal;
			  fbHomeFinish.bSofLimEnableLow:=fbHomePrepare.bSofLimEnableLowOriginal;
	        END_IF;	
          3: // restore softlimit enable
            bHomed:=FALSE;
		    bSequenceReady:=FALSE;            		            	
	        IF fbHomeFinish.bDone THEN
			  bRestoreNCDataNeeded:=FALSE;
	          bSequenceReady:=TRUE;
			  nHomingState:=0;
			  bHomed:=Axis.Status.Homed;
	        END_IF;	 
	   END_CASE;
	   
   2: // Home to high limit switch
	   CASE nHomingState OF
		  0:
		    bHomed:=Axis.Status.Homed;
            // Wait for read of velocities from NC and reset of calibration flag
	        IF fbHomePrepare.bDone AND bExecute AND NOT bSequenceReady THEN
			  bRestoreNCDataNeeded:=TRUE;
			  IF bLimitFwd THEN
                nHomingState:=1;
              ELSE
				nHomingState:=2;  //Standing on limit switch go direct to state 2 
              END_IF                                          		  
	        END_IF
		  1: // wait for reach low limit then trigger fbHomeToSwitch
		    bHomed:=FALSE;
			bSequenceReady:=FALSE;
			fbMoveVelocity.Velocity:=ABS(fbHomePrepare.fVelocityToCam);
            fbMoveVelocity.Direction:=MC_Positive_Direction;
	        bExecuteMoveVelocity:=bExecute;  // Execute MC_MoveVelocity
		    IF NOT bLimitFwd AND NOT fbMoveVelocity.Busy AND Axis.Status.NotMoving THEN //MC_MoveVelocity.Busy goes down when ramp down initiates (not ends).
			  nHomingState:=2;
		    END_IF
		  2: // Wait for fbHomeToSwitch
		    bHomed:=FALSE;
		    bSequenceReady:=FALSE;
            bExecuteMoveVelocity:=FALSE;			
            bExecuteHomeToSwitch:=TRUE;	
            fbHomeToSwitch.nSearchDirTwoardsCam:=MC_Negative_Direction;
            fbHomeToSwitch.nSearchDirOffCam:=MC_Negative_Direction;	             
	        fbHomeToSwitch.fVelocityToCamNC:=fbHomePrepare.fVelocityToCam; // High speed
  	        fbHomeToSwitch.fVelocityFromCamNC:=fbHomePrepare.fVelocityFromCam;  // Low speed              		
		    fbHomeToSwitch.bCamSensor:=NOT bLimitFwd;            	 		    
	        IF fbHomeToSwitch.bDone THEN	          
			  nHomingState:=3;
			  bExecuteFinish:=TRUE;
			  fbHomeFinish.bSofLimEnableHigh:=fbHomePrepare.bSofLimEnableHighOriginal;
			  fbHomeFinish.bSofLimEnableLow:=fbHomePrepare.bSofLimEnableLowOriginal;
	        END_IF;	
          3: // restore softlimit enable
            bHomed:=FALSE;
		    bSequenceReady:=FALSE;            		            	
	        IF fbHomeFinish.bDone THEN
			  bRestoreNCDataNeeded:=FALSE;
	          bSequenceReady:=TRUE;
			  nHomingState:=0;
			  bHomed:=Axis.Status.Homed;
	        END_IF;	 
	   END_CASE;
	   
   3: // Home on bHomeSensor via bLimitBwd
   	   CASE nHomingState OF
		  0:
		    bHomed:=Axis.Status.Homed;
            // Wait for read of velocities from NC and reset of calibration flag
	        IF fbHomePrepare.bDone AND bExecute AND NOT bSequenceReady THEN
			  bRestoreNCDataNeeded:=TRUE;
			  IF bLimitBwd THEN
                nHomingState:=1;
              ELSE
				nHomingState:=2;  //Standing on limit switch go direct to state 2 
              END_IF                                          		  
	        END_IF
		  1: // wait for reach low limit then trigger fbHomeToSwitch
		    bHomed:=FALSE;
			bSequenceReady:=FALSE;
			fbMoveVelocity.Velocity:=ABS(fbHomePrepare.fVelocityToCam);
            fbMoveVelocity.Direction:=MC_Negative_Direction;
	        bExecuteMoveVelocity:=bExecute;  // Execute MC_MoveVelocity
		    IF NOT bLimitBwd AND NOT fbMoveVelocity.Busy AND Axis.Status.NotMoving THEN //MC_MoveVelocity.Busy goes down when ramp down initiates (not ends).
			  nHomingState:=2;
		    END_IF
		  2: // Wait for fbHomeToSwitch
		    bHomed:=FALSE;
		    bSequenceReady:=FALSE;
            bExecuteMoveVelocity:=FALSE;			
            bExecuteHomeToSwitch:=TRUE;	
            fbHomeToSwitch.nSearchDirTwoardsCam:=MC_Positive_Direction;
            fbHomeToSwitch.nSearchDirOffCam:=MC_Positive_Direction;	             
	        fbHomeToSwitch.fVelocityToCamNC:=fbHomePrepare.fVelocityToCam; // High speed
  	        fbHomeToSwitch.fVelocityFromCamNC:=fbHomePrepare.fVelocityFromCam;  // Low speed              		
		    fbHomeToSwitch.bCamSensor:=bHomeSensor;            	 		    
	        IF fbHomeToSwitch.bDone THEN	          
			  nHomingState:=3;
			  bExecuteFinish:=TRUE;
			  fbHomeFinish.bSofLimEnableHigh:=fbHomePrepare.bSofLimEnableHighOriginal;
			  fbHomeFinish.bSofLimEnableLow:=fbHomePrepare.bSofLimEnableLowOriginal;
	        END_IF;	
          3: // restore softlimit enable
            bHomed:=FALSE;
		    bSequenceReady:=FALSE;            		            	
	        IF fbHomeFinish.bDone THEN
		      bRestoreNCDataNeeded:=FALSE;
	          bSequenceReady:=TRUE;
			  nHomingState:=0;
			  bHomed:=Axis.Status.Homed;
	        END_IF;	 
	   END_CASE;
	4:  // Home on bHomeSensor via bLimitFwd	   
	   CASE nHomingState OF
		  0:
		    bHomed:=Axis.Status.Homed;
            // Wait for read of velocities from NC and reset of calibration flag
	        IF fbHomePrepare.bDone AND bExecute AND NOT bSequenceReady THEN
			  bRestoreNCDataNeeded:=TRUE;
			  IF bLimitFwd THEN
                nHomingState:=1;
              ELSE
				nHomingState:=2;  //Standing on limit switch go direct to state 2 
              END_IF                                          		  
	        END_IF
		  1: // wait for reach low limit then trigger fbHomeToSwitch
		    bHomed:=FALSE;
			bSequenceReady:=FALSE;
			fbMoveVelocity.Velocity:=ABS(fbHomePrepare.fVelocityToCam);
            fbMoveVelocity.Direction:=MC_Positive_Direction;
	        bExecuteMoveVelocity:=bExecute;  // Execute MC_MoveVelocity
		    IF NOT bLimitFwd AND NOT fbMoveVelocity.Busy AND Axis.Status.NotMoving THEN //MC_MoveVelocity.Busy goes down when ramp down initiates (not ends).
			  nHomingState:=2;
		    END_IF
		  2: // Wait for fbHomeToSwitch
		    bHomed:=FALSE;
		    bSequenceReady:=FALSE;
            bExecuteMoveVelocity:=FALSE;			
            bExecuteHomeToSwitch:=TRUE;	
            fbHomeToSwitch.nSearchDirTwoardsCam:=MC_Negative_Direction;
            fbHomeToSwitch.nSearchDirOffCam:=MC_Negative_Direction;	             
	        fbHomeToSwitch.fVelocityToCamNC:=fbHomePrepare.fVelocityToCam; // High speed
  	        fbHomeToSwitch.fVelocityFromCamNC:=fbHomePrepare.fVelocityFromCam;  // Low speed              		
		    fbHomeToSwitch.bCamSensor:=bHomeSensor;            	 		    
	        IF fbHomeToSwitch.bDone THEN	          
			  nHomingState:=3;
			  bExecuteFinish:=TRUE;
			  fbHomeFinish.bSofLimEnableHigh:=fbHomePrepare.bSofLimEnableHighOriginal;
			  fbHomeFinish.bSofLimEnableLow:=fbHomePrepare.bSofLimEnableLowOriginal;
	        END_IF;	
          3: // Restore softlimit enable
            bHomed:=FALSE;
		    bSequenceReady:=FALSE;            		            	
	        IF fbHomeFinish.bDone THEN
			  bRestoreNCDataNeeded:=FALSE;
	          bSequenceReady:=TRUE;
			  nHomingState:=0;
			  bHomed:=Axis.Status.Homed;
	        END_IF;	 
	   END_CASE;
		  	    
   15: //Set current position (simplest homing sequence)
     bExecuteHomeDirect:=bExecute;
	 bHomed:=Axis.Status.Homed;
     IF fbHomeDirect.bDone THEN  //Homing ready				
	   bExecuteHomeDirect:=FALSE;				
       bSequenceReady:=TRUE;	
     END_IF	 
	 
ELSE
  fbHomeToSwitch.bCamSensor:=FALSE;
  bHomed:=Axis.Status.Homed;
END_CASE;

// Main homing block
fbHomeToSwitch(
	bExecute:=bExecuteHomeToSwitch AND bExecute AND NOT bError AND NOT bExecuteHomeDirect AND NOT bExecuteMoveVelocity,
 	bReset:=bReset,
	fHomePosition:=fHomePosition,
	Axis:=Axis
);

// Approach limit switch (error if MC_Home is used)
fbMoveVelocity(
    Execute:= bExecuteMoveVelocity AND bExecute AND NOT bError AND NOT bExecuteHomeToSwitch AND NOT bExecuteHomeDirect,
    Axis:=Axis
);

// No sequence, just set position value (nCmdDataLocal=15). Can not run if fbHomeToSwitch is executed
fbHomeDirect(
	bExecute:=bExecuteHomeDirect AND bExecute AND NOT bError  AND NOT bExecuteHomeToSwitch AND NOT bExecuteMoveVelocity,
 	bReset:=bReset,
	fHomePosition:=fHomePosition,
	Axis:=Axis
);

 
//############# Finish homing

IF NOT bexecute AND bRestoreNCDataNeeded THEN  //If homing is aborted restore is needed
	bExecuteFinish:=TRUE;
	IF fbHomeFinish.bDone THEN
	  bExecuteFinish:=FALSE;
      bRestoreNCDataNeeded:=FALSE;	
	END_IF
END_IF

fbHomeFinish(
  En:=En,
  bExecute:=bExecuteFinish,
  bReset:=bReset,
  Axis:=Axis,
);

// Error handling
IF NOT bError THEN
  IF fbHomeToSwitch.bError THEN 
	bError:=fbHomeToSwitch.bError;
	nErrorId:=fbHomeToSwitch.nErrorId;
  ELSIF fbHomeDirect.bError THEN
	bError:=fbHomeDirect.bError;
	nErrorId:=fbHomeDirect.nErrorId;
  ELSIF fbMoveVelocity.Error THEN
	bError:=fbMoveVelocity.Error;
	nErrorId:=fbMoveVelocity.ErrorId;    		    		
  END_IF;	
END_IF

// Done and busy bit
bDone:=bSequenceReady AND bExecute;
bBusy:=NOT bSequenceReady;	 

RETURN;

END_FUNCTION_BLOCK

// tc_mca_std_lib/POUs/Motion/Homing/FB_HomeToSwitch
FUNCTION_BLOCK FB_HomeToSwitch
VAR_INPUT
	En: BOOL;
	bReset: BOOL;
    bExecute: BOOL;	
    bCamSensor:BOOL;	
	nSearchDirTwoardsCam: MC_Direction;
	nSearchDirOffCam: MC_Direction;
	fHomePosition:LREAL;	
	fVelocityToCamNC: LREAL; //Velcoity when searching for cam
	fVelocityFromCamNC: LREAL; // Velocity after found cam (searching for next signal transition)
END_VAR
VAR_IN_OUT
	Axis: AXIS_REF;
END_VAR
VAR_OUTPUT
	EnO: BOOL;	
	bBusy: BOOL;
	bDone: BOOL;
	bHomed:BOOL;
	bError: BOOL;
	nErrorId: UDINT;
END_VAR
VAR
	fbHome: MC_Home;	
	fbWriteHomeDirCamToNC:FB_WriteParameterInNc_v1_00;
	fbWriteHomeDirSyncToNC:FB_WriteParameterInNc_v1_00;
	fbWriteHomeModeToNC:FB_WriteParameterInNc_v1_00;
	fbWriteHomeVelocitiesToNC: FB_HomeWriteNcVelocities;
	bConfigNCDone:BOOL:=FALSE;
	fbRTrigg: R_TRIG;
END_VAR

En:=EnO;
IF bReset THEN
	bConfigNCDone:=FALSE;
	bError:=FALSE;
	nErrorId:=0;
END_IF 
	
//Start preparation of NC if rising edge on bExecute
fbRTrigg(CLK:=bExecute);
IF fbRTrigg.Q THEN
	bConfigNCDone:=FALSE;
END_IF

 
fbWriteHomeDirCamToNC(
	bExecute:=bExecute AND NOT bConfigNCDone,
	nDeviceGroup:=16#5000,
	nIndexOffset:=16#101,	//Direction for Calibration Cam Search	
	nData:=BOOL_TO_DWORD(nSearchDirTwoardsCam=MC_Negative_Direction),//BOOL_TO_DWORD(NOT bSearchDirTwoardsCam),
	Axis:=Axis
);

fbWriteHomeDirSyncToNC(
	bExecute:= bExecute AND NOT bConfigNCDone,
	nDeviceGroup:=16#5000 ,
	nIndexOffset:=16#102 , //Direction for Sync Impuls Search
	nData:=BOOL_TO_DWORD(nSearchDirOffCam=MC_Negative_Direction),//BOOL_TO_DWORD(NOT bSearchDirOffCam),
	Axis:= Axis 
);

fbWriteHomeModeToNC(
	bExecute:=bExecute AND NOT bConfigNCDone,
	nDeviceGroup:=16#5000,
	nIndexOffset:=16#107,  //Reference Mode
	nData:=1,
	Axis:=axis);
	
fbWriteHomeVelocitiesToNC(
  En:=En,
  bExecute:=bExecute AND NOT bConfigNCDone,
  bReset:=bReset,
  fVelocityFromCam:=fVelocityFromCamNC,
  fVelocityToCam:=fVelocityToCamNC,
  Axis:=Axis);

fbHome.bCalibrationCam:=bCamSensor;

fbHome(
	Execute:=bExecute AND bConfigNCDone(* AND NOT bError*),
	Position:=fHomePosition,
	HomingMode:=0,
	Axis:=Axis
	);
bBusy:=(fbHome.Busy OR (NOT bConfigNCDone AND bExecute));
bDone:=fbHome.Done AND bConfigNCDone;
bHomed:=Axis.Status.Homed;

IF (NOT bConfigNCDone) AND fbWriteHomeDirCamToNC.bDone AND fbWriteHomeDirSyncToNC.bDone AND fbWriteHomeModeToNC.bDone AND fbWriteHomeVelocitiesToNC.bDone THEN
  bConfigNCDone:=TRUE;
END_IF

//For some reason MC_HOME gives an Error for one cycle of NC-Task 1 SVB (10ms default..) so filter with bExecute
bError:=(fbHome.Error AND bExecute) OR fbWriteHomeDirCamToNC.bError OR fbWriteHomeDirSyncToNC.bError OR fbWriteHomeModeToNC.bError OR fbWriteHomeVelocitiesToNC.bError;

IF (fbHome.Error AND bExecute) THEN
  nErrorId:=fbHome.ErrorID;
ELSIF fbWriteHomeDirCamToNC.bError THEN
  nErrorId:=fbWriteHomeDirCamToNC.nErrorId;
ELSIF fbWriteHomeDirSyncToNC.bError THEN
  nErrorId:=fbWriteHomeDirSyncToNC.nErrorId;
ELSIF fbWriteHomeModeToNC.bError THEN
  nErrorId:=fbWriteHomeModeToNC.nErrorId;
ELSIF fbWriteHomeVelocitiesToNC.bError THEN
  nErrorId:=fbWriteHomeVelocitiesToNC.nErrorId;  
END_IF

END_FUNCTION_BLOCK

// tc_mca_std_lib/POUs/ChangeConfig/FB_WriteParameterInNc_v1_00
///#########################################################
///Function block to write parameter in Nc.
///
///	Library:		
///	Tc2_MC2.lib
/// Tc2_System.lib
///
///	Global Variables:
///	
///	Data types:
///	
///	External functions:
///
///	History:
///	2014-02-05	v1.00	NB	Release code.
///
///	Known bugs:
///
///
///
///###########################################################
FUNCTION_BLOCK FB_WriteParameterInNc_v1_00
VAR_INPUT
	bExecute: BOOL;
	///16#4000=Axisdata, 16#5000=Encoderdata, 16#6000=Controldata, 16#7000=Drivedata
	nDeviceGroup: UDINT;
	nIndexOffset: UDINT;
	nData: DWORD;
END_VAR
VAR_OUTPUT
	bBusy: BOOL;
	bDone: BOOL;
	bError: BOOL;
	nErrorId: UDINT;
END_VAR
VAR_IN_OUT
	Axis: AXIS_REF;
END_VAR
VAR
	nState: UINT;
	fbADSWRITE: ADSWRITE;
END_VAR

(*Sequence to write parameter in Nc*)
CASE nState OF
0:  (*Start sequence. Wait until bExecute is TRUE*)
	IF bExecute THEN
		bBusy:=TRUE;
		bError:=FALSE;
		nErrorId:=0;
		nState:=10;
	END_IF

10: (*Write parameter in Nc*)
	fbADSWRITE(
		PORT:=500,
		IDXGRP:=nDeviceGroup+Axis.NcToPlc.AxisId,
		IDXOFFS:=nIndexOffset,
		LEN:=SIZEOF(nData),
		SRCADDR:=ADR(nData),
		WRITE:=TRUE);

	(*Wait until it's done or if an error occurs*)
	IF NOT fbADSWRITE.ERR THEN
		IF NOT fbADSWRITE.BUSY THEN
			fbADSWRITE(WRITE:=FALSE);
			nState:=20;
		END_IF
	ELSE
		nErrorId:=fbADSWRITE.ERRID;
		nState:=999;
	END_IF

20: (*Sequense is done. Waits until bExecute is FALSE*)
	bBusy:=FALSE;
	bDone:=TRUE;
	IF NOT bExecute THEN
		bDone:=FALSE;
		nState:=0;
	END_IF

999: (*Error in sequence*)
	bError:=TRUE;
	bBusy:=FALSE;
	bDone:=FALSE;
	fbADSWRITE(WRITE:=FALSE);
	IF NOT bExecute THEN
		nState:=0;
	END_IF

END_CASE

END_FUNCTION_BLOCK

// tc_mca_std_lib/POUs/Motion/Homing/FB_HomeWriteNcVelocities
FUNCTION_BLOCK FB_HomeWriteNcVelocities
VAR_INPUT
	En: BOOL;
	bReset: BOOL;
    bExecute: BOOL;		
	fVelocityToCam: LREAL;
	fVelocityFromCam: LREAL;	
END_VAR
VAR_IN_OUT
	Axis: AXIS_REF;
END_VAR
VAR_OUTPUT
	EnO: BOOL;	
	bBusy: BOOL;
	bDone: BOOL;
	bError: BOOL;
	nErrorId: UDINT;	
END_VAR
VAR
	fbExecuteRiseEdge: R_TRIG;
	fbWriteVelocityToCam:FB_WriteFloatParameter;
	fbWriteVelocityFromCam:FB_WriteFloatParameter;
END_VAR

En:=EnO;
IF bReset THEN
	bError:=FALSE;
	nErrorId:=0;
END_IF 

fbExecuteRiseEdge(CLK:=bExecute);

fbWriteVelocityToCam(
	bExecute:=bExecute,
	nDeviceGroup:= 16#4000,
	nIndexOffset:= 16#6,
	nData:=fVelocityToCam,
	Axis:= Axis);
	
fbWriteVelocityFromCam(
	bExecute:=bExecute,
	nDeviceGroup:= 16#4000,
	nIndexOffset:= 16#7,
	nData:=fVelocityFromCam,
	Axis:= Axis);

bBusy:=fbWriteVelocityFromCam.bBusy OR fbWriteVelocityToCam.bBusy;
bDone:=fbWriteVelocityFromCam.bDone AND fbWriteVelocityToCam.bDone AND bExecute;

bError:=fbWriteVelocityToCam.bError OR fbWriteVelocityFromCam.bError;
IF fbWriteVelocityToCam.bError THEN
  nErrorId:=fbWriteVelocityToCam.nErrorId;
ELSIF fbWriteVelocityFromCam.bError THEN
  nErrorId:=fbWriteVelocityFromCam.nErrorId;
END_IF

END_FUNCTION_BLOCK

// tc_mca_std_lib/POUs/ChangeConfig/FB_WriteFloatParameter
///#########################################################
///Function block to write parameter in Nc.
///
///	Library:		
///	Tc2_MC2.lib
/// Tc2_System.lib
///
///	Global Variables:
///	
///	Data types:
///	
///	External functions:
///
///	History:
///	2014-02-05	v1.00	NB	Release code.
///
///	Known bugs:
///
///
///
///###########################################################
FUNCTION_BLOCK FB_WriteFloatParameter
VAR_INPUT
	bExecute: BOOL;
	///16#4000=Axisdata, 16#5000=Encoderdata, 16#6000=Controldata, 16#7000=Drivedata
	nDeviceGroup: UDINT;
	nIndexOffset: UDINT;
	nData: LREAL;
END_VAR
VAR_OUTPUT
	bBusy: BOOL;
	bDone: BOOL;
	bError: BOOL;
	nErrorId: UDINT;
END_VAR
VAR_IN_OUT
	Axis: AXIS_REF;
END_VAR
VAR
	nState: UINT;
	fbADSWRITE: ADSWRITE;
END_VAR

(*Sequence to write parameter in Nc*)
CASE nState OF
0:  (*Start sequence. Wait until bExecute is TRUE*)
	IF bExecute THEN
		bBusy:=TRUE;
		bError:=FALSE;
		nErrorId:=0;
		nState:=10;
	END_IF

10: (*Write parameter in Nc*)
	fbADSWRITE(
		PORT:=500,
		IDXGRP:=nDeviceGroup+Axis.NcToPlc.AxisId,
		IDXOFFS:=nIndexOffset,
		LEN:=SIZEOF(nData),
		SRCADDR:=ADR(nData),
		WRITE:=TRUE);

	(*Wait until it's done or if an error occurs*)
	IF NOT fbADSWRITE.ERR THEN
		IF NOT fbADSWRITE.BUSY THEN
			fbADSWRITE(WRITE:=FALSE);
			nState:=20;
		END_IF
	ELSE
		nErrorId:=fbADSWRITE.ERRID;
		nState:=999;
	END_IF

20: (*Sequense is done. Waits until bExecute is FALSE*)
	bBusy:=FALSE;
	bDone:=TRUE;
	IF NOT bExecute THEN
		bDone:=FALSE;
		nState:=0;
	END_IF

999: (*Error in sequence*)
	bError:=TRUE;
	bBusy:=FALSE;
	bDone:=FALSE;
	fbADSWRITE(WRITE:=FALSE);
	IF NOT bExecute THEN
		nState:=0;
	END_IF

END_CASE

END_FUNCTION_BLOCK

// tc_mca_std_lib/POUs/Motion/Homing/FB_HomeDirect
FUNCTION_BLOCK FB_HomeDirect
VAR_INPUT
	En: BOOL;
	bReset: BOOL;
    bExecute: BOOL;	
	fHomePosition:LREAL;	
END_VAR
VAR_IN_OUT
	Axis: AXIS_REF;
END_VAR
VAR_OUTPUT
	EnO: BOOL;	
	bBusy: BOOL;
	bDone: BOOL;
	bHomed:BOOL;
	bError: BOOL;
	nErrorId: UDINT;
END_VAR
VAR
	fbHome: MC_Home;	
END_VAR

En:=EnO;
IF bReset THEN
	bError:=FALSE;
	nErrorId:=0;
END_IF 

fbHome(
	Execute:=bExecute,
	Position:=fHomePosition,
	HomingMode:=MC_Direct,
	bCalibrationCam:=FALSE,
	Axis:=Axis
	);
	
bBusy:=fbHome.Busy;
bDone:=fbHome.Done;
bHomed:=Axis.Status.Homed;

bError:=fbHome.Error; 

IF fbHome.Error THEN
  nErrorId:=fbHome.ErrorID;
END_IF

END_FUNCTION_BLOCK

// tc_mca_std_lib/POUs/Motion/Homing/FB_HomePrepare
FUNCTION_BLOCK FB_HomePrepare
VAR_INPUT
	En: BOOL;
	bReset: BOOL;
    bExecute: BOOL;	
    nCmdData: UINT;		
END_VAR
VAR_IN_OUT
	Axis: AXIS_REF;
END_VAR
VAR_OUTPUT
	EnO: BOOL;	
	bBusy: BOOL;
	bDone: BOOL;
	bError: BOOL;
	nErrorId: UDINT;
	bSofLimEnableLowOriginal: BOOL:=TRUE;
	bSofLimEnableHighOriginal: BOOL:=TRUE;	
	fVelocityToCam: LREAL:=0;
	fVelocityFromCam: LREAL:=0;		
END_VAR
VAR
	fbHomeReadSoftLimEnable:FB_HomeReadSoftLimEnable;	
	fbHomeDisableSoftLimEnable:FB_HomeWriteSoftLimEnable;
	fbHomeReadNCVelocities: FB_HomeReadNcVelocities;
	fbHomeResetCalibrationFlag:MC_Home;   //Only used for reset of calibration flag
	fbExecuteRiseEdge: R_TRIG;
	bExecuteReadNC:BOOL:=FALSE;
	bExecuteWriteNC:BOOL:=FALSE;
	nState:INT:=0;
END_VAR

En:=EnO;
IF bReset THEN
	bError:=FALSE;
	nErrorId:=0;
END_IF 

IF NOT bExecute THEN
  bExecuteReadNC:=FALSE;
  bExecuteWriteNC:=FALSE;   
  nState:=0;
END_IF

fbExecuteRiseEdge(CLK:=bExecute);
IF fbExecuteRiseEdge.Q THEN
  bExecuteReadNC:=TRUE;  
END_IF

// Read from NC
fbHomeReadNCVelocities(
  En:=En,
  bExecute:=bExecuteReadNC, // Actualy not needed for sequence 15 (set position only, no movement))
  bReset:=bReset,
  Axis:=Axis,
);

fbHomeReadSoftLimEnable(
	En:=En,
	bExecute:=bExecuteReadNC AND bExecute,
	Axis:=Axis,
	bReset:=bReset,	
);

// Reset calibration flag
fbHomeResetCalibrationFlag(
  Execute:=bExecuteReadNC,
  HomingMode:=MC_ResetCalibration,
  Axis:=Axis
);

bSofLimEnableLowOriginal:=fbHomeReadSoftLimEnable.bSofLimEnableLow;
bSofLimEnableHighOriginal:=fbHomeReadSoftLimEnable.bSofLimEnableHigh;	

fVelocityToCam:=fbHomeReadNCVelocities.fVelocityToCam;
fVelocityFromCam:=fbHomeReadNCVelocities.fVelocityFromCam;

IF bExecuteReadNC AND bExecute AND fbHomeReadSoftLimEnable.bDone THEN
	fbHomeDisableSoftLimEnable.bSofLimEnableHigh:=FALSE;
	fbHomeDisableSoftLimEnable.bSofLimEnableLow:=FALSE;
	bExecuteWriteNC:=TRUE; //Always write (only needed if enabled actually)
END_IF

// Write to NC (disable soft limits)
fbHomeDisableSoftLimEnable(
	En:=En,
	bExecute:=bExecuteWriteNC AND bExecute,
	Axis:=Axis,
	bReset:=bReset,	
);

bBusy:=fbHomeReadSoftLimEnable.bBusy OR fbHomeDisableSoftLimEnable.bBusy OR fbHomeReadNCVelocities.bBusy OR fbHomeResetCalibrationFlag.Busy;
bDone:=fbHomeReadSoftLimEnable.bDone AND fbHomeDisableSoftLimEnable.bDone AND fbHomeReadNCVelocities.bDone AND fbHomeResetCalibrationFlag.Done AND bExecute;

bError:=fbHomeReadSoftLimEnable.bError OR fbHomeDisableSoftLimEnable.bError OR fbHomeReadNCVelocities.bError OR fbHomeResetCalibrationFlag.Error;
IF fbHomeReadSoftLimEnable.bError THEN
  nErrorId:=fbHomeReadSoftLimEnable.nErrorId;
ELSIF fbHomeDisableSoftLimEnable.bError THEN
  nErrorId:=fbHomeDisableSoftLimEnable.nErrorId;
ELSIF fbHomeResetCalibrationFlag.Error THEN
  nErrorId:=fbHomeResetCalibrationFlag.ErrorId;
END_IF

END_FUNCTION_BLOCK

// tc_mca_std_lib/POUs/Motion/Homing/FB_HomeReadSoftLimEnable
FUNCTION_BLOCK FB_HomeReadSoftLimEnable
VAR_INPUT
	En: BOOL;
	bReset: BOOL;
    bExecute: BOOL;			
END_VAR
VAR_IN_OUT
	Axis: AXIS_REF;
END_VAR
VAR_OUTPUT
	EnO: BOOL;	
	bBusy: BOOL;
	bDone: BOOL;
	bError: BOOL;
	nErrorId: UDINT;	
	bSofLimEnableLow: BOOL:=TRUE;
	bSofLimEnableHigh: BOOL:=TRUE;
END_VAR
VAR
	fbReadSoftLimEnableLow:FB_ReadParameterInNc_v1_00;
	fbReadSoftLimEnableHigh:FB_ReadParameterInNc_v1_00;
END_VAR

En:=EnO;
IF bReset THEN
	bError:=FALSE;
	nErrorId:=0;
END_IF 
	
fbReadSoftLimEnableLow(
	bExecute:=bExecute,
	nDeviceGroup:= 16#5000,
	nIndexOffset:= 16#B,
	Axis:= Axis);

fbReadSoftLimEnableHigh(
	bExecute:=bExecute,
	nDeviceGroup:= 16#5000,
	nIndexOffset:= 16#C,
	Axis:= Axis);
	
bSofLimEnableLow:=DWORD_TO_BOOL(fbReadSoftLimEnableLow.nData);
bSofLimEnableHigh:=DWORD_TO_BOOL(fbReadSoftLimEnableHigh.nData);	

bBusy:=fbReadSoftLimEnableLow.bBusy OR fbReadSoftLimEnableHigh.bBusy;
bDone:=fbReadSoftLimEnableLow.bDone AND fbReadSoftLimEnableHigh.bDone AND bExecute;

bError:=fbReadSoftLimEnableLow.bError OR fbReadSoftLimEnableHigh.bError;
IF fbReadSoftLimEnableLow.bError THEN
  nErrorId:=fbReadSoftLimEnableLow.nErrorId;
ELSIF fbReadSoftLimEnableHigh.bError THEN
  nErrorId:=fbReadSoftLimEnableHigh.nErrorId;
END_IF

END_FUNCTION_BLOCK

// tc_mca_std_lib/POUs/ChangeConfig/FB_ReadParameterInNc_v1_00
///#########################################################
///Function block to read parameter in Nc.
///
///	Library:		
///	Tc2_MC2.lib
/// Tc2_System.lib
///
///	Global Variables:
///	
///	Data types:
///	
///	External functions:
///
///	History:
///	2014-02-05	v1.00	NB	Release code.
///
///	Known bugs:
///
///
///
///###########################################################
FUNCTION_BLOCK FB_ReadParameterInNc_v1_00
VAR_INPUT
	bExecute: BOOL;
	///16#4000=Axisdata, 16#5000=Encoderdata, 16#6000=Controldata, 16#7000=Drivedata
	nDeviceGroup: UDINT;
	nIndexOffset: UDINT;
END_VAR
VAR_OUTPUT
	nData: DWORD;
	bBusy: BOOL;
	bDone: BOOL;
	bError: BOOL;
	nErrorId: UDINT;
END_VAR
VAR_IN_OUT
	Axis: AXIS_REF;
END_VAR
VAR
	nState: UINT;
	fbADSREAD: ADSREAD;
END_VAR

(*Sequence to read parameter in Nc*)
CASE nState OF
0:  (*Start sequence. Wait until bExecute is TRUE*)
	IF bExecute THEN
		bBusy:=TRUE;
		bError:=FALSE;
		nErrorId:=0;
		nState:=10;
	END_IF

10: (*Read parameter in Nc*)
	fbADSREAD(
		PORT:=500,
		IDXGRP:=nDeviceGroup+Axis.NcToPlc.AxisId,
		IDXOFFS:=nIndexOffset,
		LEN:=SIZEOF(nData),
		DESTADDR:=ADR(nData),
		READ:=TRUE);

	(*Wait until it's done or if an error occurs*)
	IF NOT fbADSREAD.ERR THEN
		IF NOT fbADSREAD.BUSY THEN
			fbADSREAD(READ:=FALSE);
			nState:=20;
		END_IF
	ELSE
		nErrorId:=fbADSREAD.ERRID;
		nState:=999;
	END_IF

20: (*Sequense is done. Waits until bExecute is FALSE*)
	bBusy:=FALSE;
	bDone:=TRUE;
	IF NOT bExecute THEN
		bDone:=FALSE;
		nState:=0;
	END_IF

999: (*Error in sequence*)
	bError:=TRUE;
	bBusy:=FALSE;
	bDone:=FALSE;
	fbADSREAD(READ:=FALSE);
	IF NOT bExecute THEN
		nState:=0;
	END_IF

END_CASE

END_FUNCTION_BLOCK

// tc_mca_std_lib/POUs/Motion/Homing/FB_HomeWriteSoftLimEnable
FUNCTION_BLOCK FB_HomeWriteSoftLimEnable
VAR_INPUT
	En: BOOL;
	bReset: BOOL;
    bExecute: BOOL;		
	bSofLimEnableLow: BOOL:=TRUE;
	bSofLimEnableHigh: BOOL:=TRUE;
END_VAR
VAR_IN_OUT
	Axis: AXIS_REF;
END_VAR
VAR_OUTPUT
	EnO: BOOL;	
	bBusy: BOOL;
	bDone: BOOL;
	bError: BOOL;
	nErrorId: UDINT;	
END_VAR
VAR
	fbExecuteRiseEdge: R_TRIG;
	fbWriteSoftLimEnableLow:FB_WriteParameterInNc_v1_00;
	fbWriteSoftLimEnableHigh:FB_WriteParameterInNc_v1_00;
END_VAR

En:=EnO;
IF bReset THEN
	bError:=FALSE;
	nErrorId:=0;
END_IF 

fbExecuteRiseEdge(CLK:=bExecute);

fbWriteSoftLimEnableLow(
	bExecute:=bExecute,
	nDeviceGroup:= 16#5000,
	nIndexOffset:= 16#B,
	nData:=BOOL_TO_DWORD(bSofLimEnableLow),
	Axis:= Axis);
	
fbWriteSoftLimEnableHigh(
	bExecute:=bExecute,
	nDeviceGroup:= 16#5000,
	nIndexOffset:= 16#C,
	nData:=BOOL_TO_DWORD(bSofLimEnableHigh),
	Axis:= Axis);

bBusy:=fbWriteSoftLimEnableLow.bBusy OR fbWriteSoftLimEnableHigh.bBusy;
bDone:=fbWriteSoftLimEnableLow.bDone AND fbWriteSoftLimEnableHigh.bDone AND bExecute;

bError:=fbWriteSoftLimEnableHigh.bError OR fbWriteSoftLimEnableLow.bError;
IF fbWriteSoftLimEnableHigh.bError THEN
  nErrorId:=fbWriteSoftLimEnableHigh.nErrorId;
ELSIF fbWriteSoftLimEnableLow.bError THEN
  nErrorId:=fbWriteSoftLimEnableLow.nErrorId;
END_IF

END_FUNCTION_BLOCK

// tc_mca_std_lib/POUs/Motion/Homing/FB_HomeReadNcVelocities
FUNCTION_BLOCK FB_HomeReadNcVelocities
VAR_INPUT
	En: BOOL;
	bReset: BOOL;
    bExecute: BOOL;			
END_VAR
VAR_IN_OUT
	Axis: AXIS_REF;
END_VAR
VAR_OUTPUT
	EnO: BOOL;	
	bBusy: BOOL;
	bDone: BOOL;
	bError: BOOL;
	nErrorId: UDINT;	
	fVelocityToCam: LREAL;
	fVelocityFromCam: LREAL;
END_VAR
VAR
	fbReadVelocityToCam:FB_ReadFloatParameter;
	fbReadVelocityFromCam:FB_ReadFloatParameter;
END_VAR

En:=EnO;
IF bReset THEN
	bError:=FALSE;
	nErrorId:=0;
END_IF 
	
fbReadVelocityToCam(
	bExecute:=bExecute,
	nDeviceGroup:= 16#4000,
	nIndexOffset:= 16#6,
	Axis:= Axis);
	
fbReadVelocityFromCam(
	bExecute:=bExecute,
	nDeviceGroup:= 16#4000,
	nIndexOffset:= 16#7,
	Axis:= Axis);
	
fVelocityToCam:=fbReadVelocityToCam.nData;
fVelocityFromCam:=fbReadVelocityFromCam.nData;	

bBusy:=fbReadVelocityFromCam.bBusy OR fbReadVelocityToCam.bBusy;
bDone:=fbReadVelocityFromCam.bDone AND fbReadVelocityToCam.bDone AND bExecute;

bError:=fbReadVelocityToCam.bError OR fbReadVelocityFromCam.bError;
IF fbReadVelocityToCam.bError THEN
  nErrorId:=fbReadVelocityToCam.nErrorId;
ELSIF fbReadVelocityFromCam.bError THEN
  nErrorId:=fbReadVelocityFromCam.nErrorId;
END_IF

END_FUNCTION_BLOCK

// tc_mca_std_lib/POUs/ChangeConfig/FB_ReadFloatParameter
FUNCTION_BLOCK FB_ReadFloatParameter
VAR_INPUT
	bExecute: BOOL;
	///16#4000=Axisdata, 16#5000=Encoderdata, 16#6000=Controldata, 16#7000=Drivedata
	nDeviceGroup: UDINT;
	nIndexOffset: UDINT;
END_VAR
VAR_OUTPUT
	nData: LREAL;
	bBusy: BOOL;
	bDone: BOOL;
	bError: BOOL;
	nErrorId: UDINT;
END_VAR
VAR_IN_OUT
	Axis: AXIS_REF;
END_VAR
VAR
	nState: UINT;
	fbADSREAD: ADSREAD;
END_VAR

(*Sequence to read parameter in Nc*)
CASE nState OF
0:  (*Start sequence. Wait until bExecute is TRUE*)
	IF bExecute THEN
		bBusy:=TRUE;
		bError:=FALSE;
		nErrorId:=0;
		nState:=10;
	END_IF

10: (*Read parameter in Nc*)
	fbADSREAD(
		PORT:=500,
		IDXGRP:=nDeviceGroup+Axis.NcToPlc.AxisId,
		IDXOFFS:=nIndexOffset,
		LEN:=SIZEOF(nData),
		DESTADDR:=ADR(nData),
		READ:=TRUE);

	(*Wait until it's done or if an error occurs*)
	IF NOT fbADSREAD.ERR THEN
		IF NOT fbADSREAD.BUSY THEN
			fbADSREAD(READ:=FALSE);
			nState:=20;
		END_IF
	ELSE
		nErrorId:=fbADSREAD.ERRID;
		nState:=999;
	END_IF

20: (*Sequense is done. Waits until bExecute is FALSE*)
	bBusy:=FALSE;
	bDone:=TRUE;
	IF NOT bExecute THEN
		bDone:=FALSE;
		nState:=0;
	END_IF

999: (*Error in sequence*)
	bError:=TRUE;
	bBusy:=FALSE;
	bDone:=FALSE;
	fbADSREAD(READ:=FALSE);
	IF NOT bExecute THEN
		nState:=0;
	END_IF

END_CASE

END_FUNCTION_BLOCK

// tc_mca_std_lib/POUs/Motion/Homing/FB_HomeFinish
FUNCTION_BLOCK FB_HomeFinish
VAR_INPUT
	En: BOOL;
	bReset: BOOL;
    bExecute: BOOL;	
    nCmdData: UINT;
	bSofLimEnableLow: BOOL:=TRUE;
	bSofLimEnableHigh: BOOL:=TRUE;			
END_VAR
VAR_IN_OUT
	Axis: AXIS_REF;
END_VAR
VAR_OUTPUT
	EnO: BOOL;	
	bBusy: BOOL;
	bDone: BOOL;
	bError: BOOL;
	nErrorId: UDINT;
END_VAR
VAR		
	fbHomewriteSoftLimEnable:FB_HomeWriteSoftLimEnable;	
	fbExecuteRiseEdge: R_TRIG;	
	bExecuteWriteNC:BOOL:=FALSE;
	nState:INT:=0;
END_VAR

En:=EnO;
IF bReset THEN
	bError:=FALSE;
	nErrorId:=0;
END_IF 

IF NOT bExecute THEN
  bExecuteWriteNC:=FALSE;
  fbHomewriteSoftLimEnable.bSofLimEnableLow:=bSofLimEnableLow;
  fbHomewriteSoftLimEnable.bSofLimEnableHigh:=bSofLimEnableHigh;   
  nState:=0;
END_IF

fbExecuteRiseEdge(CLK:=bExecute);
IF fbExecuteRiseEdge.Q THEN
  bExecuteWriteNC:=TRUE;  
  fbHomewriteSoftLimEnable.bSofLimEnableLow:=bSofLimEnableLow;
  fbHomewriteSoftLimEnable.bSofLimEnableHigh:=bSofLimEnableHigh;
END_IF

// Write to NC (disable soft limits)
fbHomewriteSoftLimEnable(
	En:=En,
	bExecute:=bExecuteWriteNC AND bExecute,
	Axis:=Axis,
	bReset:=bReset,	
);

bBusy:=fbHomewriteSoftLimEnable.bBusy;
bDone:=fbHomewriteSoftLimEnable.bDone;

bError:=fbHomewriteSoftLimEnable.bError;
IF fbHomewriteSoftLimEnable.bError THEN
  nErrorId:=fbHomewriteSoftLimEnable.nErrorId;
END_IF

END_FUNCTION_BLOCK

// POUs/Motion/FB_SetEnables
FUNCTION_BLOCK FB_SetEnables
VAR_IN_OUT
	stMotionStage: DUT_MotionStage;
END_VAR

stMotionStage.bAllForwardEnable := stMotionStage.bLimitForwardEnable AND (stMotionStage.bGantryForwardEnable OR NOT stMotionStage.bGantryAxis);
stMotionStage.bAllBackwardEnable := stMotionStage.bLimitBackwardEnable AND (stMotionStage.bGantryBackwardEnable OR NOT stMotionStage.bGantryAxis);

stMotionStage.bAllEnable := stMotionStage.bEnable AND stMotionStage.bHardwareEnable;

END_FUNCTION_BLOCK

// POUs/Motion/FB_StatePTPMove
FUNCTION_BLOCK FB_StatePTPMove
// For your pytmc pragma on this block, specify io accordingly:
// 1. use input or i if you want the set position to be immutable
// 2. use io if you want to set position to be mutable from epics
VAR_INPUT
	{attribute 'pytmc' := '
		pv: INFO
	'}
	stPositionState: DUT_PositionState;
	
	{attribute 'pytmc' := '
		pv: EXEC
		io: io
	'}
	bExecute: BOOL;
	
	{attribute 'pytmc' := '
		pv: MPS_OK
		io: input
	'}
	bMPSOk: BOOL;
	
	{attribute 'pytmc' := '
		pv: EPS_OK
		io: input
	'}
	bEPSOk: BOOL;
END_VAR
VAR_IN_OUT
	stMotionStage: DUT_MotionStage;
END_VAR
VAR_OUTPUT
	{attribute 'pytmc' := '
		pv: AT_STATE
		io: input
	'}
	bAtState: BOOL;
	
	{attribute 'pytmc' := '
		pv: DMOV
		io: input
	'}
	bDone: BOOL;
	
	{attribute 'pytmc' := '
		pv: BUSY
		io: input
	'}
	bBusy: BOOL;
	
	{attribute 'pytmc' := '
		pv: ERR
		io: input
	'}
	bError: BOOL;
	
	{attribute 'pytmc' := '
		pv: ERRMsg
		io: input
	'}
	sError: STRING;
END_VAR
VAR
	bExecTrig: R_TRIG;
	bExecEnd: F_TRIG;
	fActPosition: LREAL;
	fLowPos: LREAL;
	fHighPos: LREAL;
END_VAR

bExecTrig(CLK:=bExecute);
IF bExecTrig.Q AND bMPSOk AND bEPSOk THEN
	IF NOT stMotionStage.bBusy AND NOT stMotionStage.bError THEN
		stMotionStage.bExecute := TRUE;
		stMotionStage.nCommand := ENUM_EpicsMotorCmd.EPICS_MOTOR_MOVE_ABS;
		stMotionStage.fPosition := stPositionState.fPosition;
		stMotionStage.fVelocity := stPositionState.fVelocity;
		stMotionStage.fAcceleration := stPositionState.fAccel;
		stMotionStage.fDeceleration := stPositionState.fDecel;
		bDone := FALSE;
		bBusy := TRUE;
	END_IF
END_IF
bError := stMotionStage.bError;
sError := stMotionStage.sErrorMessage;

fActPosition := stMotionStage.stAxisStatus.fActPosition;
fLowPos := stPositionState.fPosition - stPositionState.fDelta;
fHighPos := stPositionState.fPosition + stPositionState.fDelta;
IF (fLowPos < fActPosition) AND (fHighPos > fActPosition) THEN
	bAtState := TRUE;
	IF NOT stMotionStage.bBusy THEN
		bDone := TRUE;
		bBusy := FALSE;
		bExecute := FALSE;
	END_IF
ELSE
	bAtState := FALSE;
END_IF

bExecEnd(CLK:=bExecute);
IF bExecEnd.Q AND bBusy THEN
	stMotionStage.bExecute := FALSE;
END_IF

IF NOT stMotionStage.bExecute OR NOT bExecute THEN
	bDone := TRUE;
	bBusy := FALSE;
	bExecute := FALSE;
END_IF

END_FUNCTION_BLOCK

// POUs/MotorTesting/FB_MicroStepCountTest
FUNCTION_BLOCK FB_MicroStepCountTest
VAR_INPUT
	bExecute: BOOL;
	fStepSize: LREAL;
	nSteps: UINT;
	fMicroStep: LREAL;
	fVelocity: LREAL;
	tSettleTime: TIME;
END_VAR
VAR_IN_OUT
	Axis: AXIS_REF;
END_VAR
VAR_OUTPUT
	nStepsCounted: UINT;
	nTheorySteps: UINT;
	fPercent: LREAL;
	fEstMicroSize: LREAL;
END_VAR
VAR
	fbMoveRel: MC_MoveRelative;
	fbSettleTimer: TON;
	bDoMove: BOOL;
	nStepCounter: UINT;
	
	arrPosBuffer: ARRAY [0..99] OF LREAL;
	fAvgPos: LREAL;
	nArrIndex: UINT;
	nLoopIndex: UINT;
	
	fStartPos: LREAL;
	fPrevPos: LREAL;
	fStepChange: LREAL;
	
	fStepSum: LREAL;
END_VAR

// Motion FB
fbMoveRel(Axis:=Axis,
	Execute:=bDoMove,
	Distance:=fStepSize,
	Velocity:=fVelocity);
	
// Settle time
fbSettleTimer(IN:=fbMoveRel.Done,
	PT:=tSettleTime);
	
// Re-enable the move for next cycle
bDoMove := bExecute AND nStepCounter < nSteps;

// Calculate rolling average
arrPosBuffer[nArrIndex] := Axis.NcToPlc.ActPos;
fAvgPos := 0;
FOR nLoopIndex := 0 TO 99 DO
	fAvgPos := fAvgPos + arrPosBuffer[nLoopIndex];
END_FOR;
fAvgPos := fAvgPos / 100;
nArrIndex := (nArrIndex + 1) MOD 100;

// Initialize starting variables
IF NOT bExecute THEN
	fStartPos := fAvgPos;
	fPrevPos := fAvgPos;
END_IF

// Check results
IF fbSettleTimer.Q THEN
	fStepChange := fAvgPos - fPrevPos;
	// Invert fStepChange if we were doing negative steps
	IF fStepSize < 0 THEN
		fStepChange := fStepChange * -1;
	END_IF
	IF fStepChange > fMicroStep * 0.5 THEN
		nStepsCounted := nStepsCounted + 1;
		fStepSum := fStepSum + fStepChange;
		fEstMicroSize := fStepSum / nStepsCounted;
	END_IF
	nTheorySteps := DINT_TO_UINT(TRUNC(ABS((fStartPos - fAvgPos) / fMicroStep)));
	IF nTheorySteps > 0 THEN
		fPercent := 100 * nStepsCounted / nTheorySteps;
	END_IF
	fPrevPos := fAvgPos;
	nStepCounter := nStepCounter + 1;
	// Reset the move block
	bDoMove := FALSE;
END_IF

END_FUNCTION_BLOCK

// tc_mca_std_lib/POUs/ErrorHandling/FB_ErrorList
FUNCTION_BLOCK FB_ErrorList

VAR_INPUT
	En : BOOL;											//Enable input
	bReset : BOOL;										//Delete all Error entry
	lErrorID : ULINT;									//ErrorID to be acknoledged
	bACK : BOOL;										//Acknoledge the given error and delete it from the list
END_VAR
	
VAR_OUTPUT
	EnO : BOOL;											//Enable output
	nNoError: UINT;										//Number of Errors
	nNoOverflow : INT;									//Number of Overflows
	pErrorSystem : POINTER TO ST_ErrorSystem;			//Pointer to ErrorSystem
END_VAR

VAR
	nFreePos : UINT;									//Number of free position in the list
	nListCnt1 : UINT;									//work variable
	ErrorSystem : ST_ErrorSystem;						//Data structure of the Error list
END_VAR

(*
* ================================================================================
*                                   DESCRIPTION
* ================================================================================
* This Function Block implements the core structure of the Error/Warning Handling
* system. It realizes the datastructure containing every Error Entry, collect
* statistics about the usage and manage the Error Entries.
* Note: The system is under development, most of the functionalities are not
* implemented or existing functionalities may change with time.
* ================================================================================
*)
EnO := En;

//Ponter to ErrorSystem
pErrorSystem := ADR(ErrorSystem);

//Number of overflows
nNoOverflow := ErrorSystem.nNoOverflows;

IF bReset THEN
	MEMSET ( ADR(ErrorSystem.aErrorData[0]), 0, GVL_ErrorSystem.cSizeOfErrorData * SIZEOF(DUT_TerminalError));
	ErrorSystem.lNextErrorID := 1;
END_IF

//Number of errors in the system
nNoError := 0;
FOR nListCnt1 := 0 TO GVL_ErrorSystem.cSizeOfErrorData - 1 DO
	IF ErrorSystem.aErrorData[nListCnt1].Error_ID <> 0  THEN
		nNoError := nNoError+1; 
	END_IF
END_FOR
ErrorSystem.nNoErrors := nNoError;

//Number of free position in the list
nFreePos := GVL_ErrorSystem.cSizeOfErrorData - nNoError;

//Acknoledge specified Error entry
IF bACK THEN
	FOR nListCnt1 := 0 TO GVL_ErrorSystem.cSizeOfErrorData - 1 DO
		IF ErrorSystem.aErrorData[nListCnt1].Error_ID = lErrorID THEN
			ErrorSystem.aErrorData[nListCnt1].ErrorState := DUT_ErrorState.Acknowledged;
		END_IF
	END_FOR
END_IF

//Deleting acknoledged errors
FOR nListCnt1 := 0 TO GVL_ErrorSystem.cSizeOfErrorData - 1 DO
	IF ErrorSystem.aErrorData[nListCnt1].ErrorState = DUT_ErrorState.Acknowledged THEN
		MEMMOVE (ADR(ErrorSystem.aErrorData[nListCnt1]), ADR(ErrorSystem.aErrorData[nListCnt1+1]), (GVL_ErrorSystem.cSizeOfErrorData - 1 - nListCnt1) * SIZEOF(DUT_TerminalError));
		MEMSET(ADR(ErrorSystem.aErrorData[GVL_ErrorSystem.cSizeOfErrorData - 1]), 0, SIZEOF(DUT_TerminalError));
	END_IF
END_FOR

END_FUNCTION_BLOCK

// tc_mca_std_lib/POUs/ErrorHandling/FB_TerminalError
FUNCTION_BLOCK FB_TerminalError

VAR_INPUT
	En					: BOOL;
	iTerminal_ID		: INT;
	bWcState			: BOOL;
	uiInfoData_State	: UINT;
	pErrorSystem		: POINTER TO ST_ErrorSystem;					//Pointer to the error system
END_VAR

VAR_OUTPUT
	EnO : BOOL;
	bError : BOOL := FALSE;
END_VAR

VAR
	iStateError : UINT;
	iOtherError : UINT;
	ErrorData	: DUT_TerminalError;
	nErrSysCNT	: UINT;
	
	//testing
	bStateChanged : BOOL;						//Indicate if state change happened
	uiInfoData_State_Prev : UINT := 16#8;		//Previous value of Infodata.State
	bWcState_Prev : BOOL := FALSE;				//Previous state of WcState
	
	//FB-s
	
END_VAR

(*
Currently:

Problem:

TODO:

*)

//Connect EN to EnO
EnO:=En;

//Check if pointer is OK
IF pErrorSystem=0 THEN RETURN; END_IF

//Any difference from normal state creates an error
IF En AND (bWcState OR uiInfoData_State<>16#8) THEN
	bError:=TRUE;
ELSE
	bError:=FALSE;
END_IF

//Change detection
IF uiInfoData_State <> uiInfoData_State_Prev OR bWcState <> bWcState_Prev THEN
	bStateChanged := TRUE;
ELSE
	bStateChanged := FALSE;
END_IF

//Update previous values
uiInfoData_State_Prev := uiInfoData_State;
bWcState_Prev := bWcState;

//Decision tree
IF bStateChanged THEN
	IF bError THEN
		IF ErrorData.ErrorState = DUT_ErrorState.Active THEN
			//Close active error
			//Read system time
			ErrorData.nDateTimeOff := Tc2_EtherCAT.F_GetActualDcTime64();
			ErrorData.sDateTimeOff := Tc2_EtherCat.DCTIME64_TO_STRING(ErrorData.nDateTimeOff);
			ErrorData.ErrorState := DUT_ErrorState.Inactive;
			//Write Off-time to Error System
			FOR nErrSysCNT := 0 TO GVL_ErrorSystem.cSizeOfErrorData - 1 DO
				IF pErrorSystem^.aErrorData[nErrSysCNT].Error_ID = ErrorData.Error_ID THEN
					pErrorSystem^.aErrorData[nErrSysCNT].nDateTimeOff := ErrorData.nDateTimeOff;
					pErrorSystem^.aErrorData[nErrSysCNT].sDateTimeOff := ErrorData.sDateTimeOff;
					pErrorSystem^.aErrorData[nErrSysCNT].ErrorState := DUT_ErrorState.Inactive;
					EXIT;
				END_IF
			END_FOR
				
			//Clear ErrorData
			MEMSET(ADR(ErrorData), 0, SIZEOF(ErrorData));
		END_IF
		
		//Open a new error
		ErrorData.ErrorState := DUT_ErrorState.Active;												//Set Error State
		ErrorData.nDateTimeOn := Tc2_EtherCAT.F_GetActualDcTime64();								//Get system time
		ErrorData.sDateTimeOn := Tc2_EtherCat.DCTIME64_TO_STRING(ErrorData.nDateTimeOn);			//Convert to string
		ErrorData.iTerminalID := iTerminal_ID;														//Terminal_ID
		ErrorData.bWcState := bWcState;																//WcState bit
		ErrorData.uiInfoDataState := uiInfoData_State;												//uiInfoData_State
		
		//Error message according to uiInfoData_State and WcState
		iStateError := (uiInfoData_State AND 16#000F);												//Mask for operation state 
		iOtherError := (uiInfoData_State AND 16#00F0);												//Mask for the other 3 kind of errors
		//Error messages according to the least significant digit
		CASE iStateError OF
			16#0001 : ErrorData.sErrorMessage := 'Slave in INIT state;   ';
			16#0002 : ErrorData.sErrorMessage := 'Slave in PREOP state;   ';
			16#0003 : ErrorData.sErrorMessage := 'Slave in BOOT state;   ';
			16#0004 : ErrorData.sErrorMessage := 'Slave in SAFEOP state;   ';
			16#0008 : ;																			//Normal operation state
		ELSE
			ErrorData.sErrorMessage := 'Undefined State of operation;   ';						//I hope we will never see this message
			ErrorData.sErrorMessage := CONCAT (ErrorData.sErrorMessage, UINT_TO_STRING(iStateError));
			ErrorData.sErrorMessage := CONCAT (ErrorData.sErrorMessage, '   ');
		END_CASE
		
		//Error messages according to the second least significant digit
		CASE iOtherError OF
			16#0000 : ;																			//No error case
			16#0010 : ErrorData.sErrorMessage := CONCAT (ErrorData.sErrorMessage, 'Slave signals error;   ');
			16#0020 : ErrorData.sErrorMessage := CONCAT (ErrorData.sErrorMessage, 'Invalid vendorID/productCode read;   ');
			16#0040 : ErrorData.sErrorMessage := CONCAT (ErrorData.sErrorMessage, 'Initialisation error occured;   ');
		ELSE
			ErrorData.sErrorMessage := CONCAT (ErrorData.sErrorMessage, 'Undefined Error ID: ');
			ErrorData.sErrorMessage := CONCAT (ErrorData.sErrorMessage, UINT_TO_STRING(iOtherError));
			ErrorData.sErrorMessage := CONCAT (ErrorData.sErrorMessage, '   ');
		END_CASE
	
		//Errormessage according to WcState bit
		IF bWcState THEN
			ErrorData.sErrorMessage := CONCAT (ErrorData.sErrorMessage, 'Invalid Data;');
		END_IF
		
		//Check for overflow
		IF pErrorSystem^.nNoErrors = GVL_ErrorSystem.cSizeOfErrorData THEN
			pErrorSystem^.nNoOverflows := pErrorSystem^.nNoOverflows+1;
		END_IF
		
		//Write Error Data into Error System
		ErrorData.Error_ID := pErrorSystem^.lNextErrorID ;
		MEMMOVE( ADR(pErrorSystem^.aErrorData[1]), ADR(pErrorSystem^.aErrorData[0]), (GVL_ErrorSystem.cSizeOfErrorData-1) * SIZEOF(DUT_TerminalError));
		pErrorSystem^.aErrorData[0] := ErrorData;
		pErrorSystem^.lNextErrorID := pErrorSystem^.lNextErrorID+1;
		
	ELSE
		//Close Active Error
		//Read system time
		ErrorData.nDateTimeOff := Tc2_EtherCAT.F_GetActualDcTime64();
		ErrorData.sDateTimeOff := Tc2_EtherCat.DCTIME64_TO_STRING(ErrorData.nDateTimeOff);
		ErrorData.ErrorState := DUT_ErrorState.Inactive;
		
		//Write Off time to Error System
		FOR nErrSysCNT := 0 TO GVL_ErrorSystem.cSizeOfErrorData - 1 DO
			IF pErrorSystem^.aErrorData[nErrSysCNT].Error_ID = ErrorData.Error_ID THEN
				pErrorSystem^.aErrorData[nErrSysCNT].nDateTimeOff := ErrorData.nDateTimeOff;
				pErrorSystem^.aErrorData[nErrSysCNT].sDateTimeOff := ErrorData.sDateTimeOff;
				pErrorSystem^.aErrorData[nErrSysCNT].ErrorState := DUT_ErrorState.Inactive;
				EXIT;
			END_IF
		END_FOR
			
		//Clear ErrorData
		MEMSET(ADR(ErrorData), 0, SIZEOF(ErrorData));
	END_IF
END_IF

END_FUNCTION_BLOCK

// tc_mca_std_lib/POUs/Hardware/EtherCAT_Terminals/Analog_Inputs/EL3174_0002
//EL3174-0002 | 4-channel analog input, -10/0...+10V, -20/0/+4...20mA, 16 bit, differential
FUNCTION_BLOCK EL3174_0002

VAR_INPUT
	En: BOOL;
	iTerminal_ID : INT;
	ErrorSystem : POINTER TO ST_ErrorSystem;
END_VAR
	
VAR_OUTPUT
	EnO: BOOL;
	iAi_Ch1_Value : INT;
	iAi_Ch2_Value : INT;
	iAi_Ch3_Value : INT;
	iAi_Ch4_Value : INT;
	bError: BOOL;
END_VAR

VAR
	//Channels
	AI_Std_Ch_1_Status	AT %I* : WORD;
	AI_Std_Ch_1_Value 	AT %I* : INT;
	AI_Std_Ch_2_Status 	AT %I* : WORD;
	AI_Std_Ch_2_Value 	AT %I* : INT;
	AI_Std_Ch_3_Status 	AT %I* : WORD;
	AI_Std_Ch_3_Value 	AT %I* : INT;
	AI_Std_Ch_4_Status 	AT %I* : WORD;
	AI_Std_Ch_4_Value 	AT %I* : INT;
	
	//Terminal status
	WcState_WcState AT %I*: BOOL;
	InfoData_State AT %I*: UINT;
	
	//FB-s
	EL3174_0002_Error : FB_TerminalError;
END_VAR

(*
* TODO:
* Status words of the channels
*)

EnO := En;

//Error FB instance
EL3174_0002_Error(
	En := TRUE,
	iTerminal_ID := iTerminal_ID,
	bWcState := WcState_WcState,
	uiInfoData_State := InfoData_State,
	pErrorSystem := ErrorSystem,
	bError => bError,
);

IF En THEN
	IF bError = FALSE THEN
		iAi_Ch1_Value := AI_Std_Ch_1_Value;
		iAi_Ch2_Value := AI_Std_Ch_2_Value;
		iAi_Ch3_Value := AI_Std_Ch_3_Value;
		iAi_Ch4_Value := AI_Std_Ch_4_Value;
	ELSE
		iAi_Ch1_Value := 0;
		iAi_Ch2_Value := 0;
		iAi_Ch3_Value := 0;
		iAi_Ch4_Value := 0;
	END_IF
END_IF

END_FUNCTION_BLOCK

// tc_mca_std_lib/POUs/Hardware/EtherCAT_Terminals/Analog_Inputs/EL3214
//EL3214 | 4-channel analog input terminal, PT100 (RTD)
FUNCTION_BLOCK EL3214

VAR_INPUT
	En: BOOL;
	iTerminal_ID : INT;
	ErrorSystem : POINTER TO ST_ErrorSystem;
END_VAR

VAR_OUTPUT
	EnO: BOOL;
	iAi_Ch1_Value : INT;
	iAi_Ch2_Value : INT;
	iAi_Ch3_Value : INT;
	iAi_Ch4_Value : INT;
	bError: BOOL;
END_VAR

VAR
	//Channels
	AI_RTD_Ch_1_Status	AT %I* : WORD;
	AI_RTD_Ch_1_Value 	AT %I* : INT;
	AI_RTD_Ch_2_Status 	AT %I* : WORD;
	AI_RTD_Ch_2_Value 	AT %I* : INT;
	AI_RTD_Ch_3_Status 	AT %I* : WORD;
	AI_RTD_Ch_3_Value 	AT %I* : INT;
	AI_RTD_Ch_4_Status 	AT %I* : WORD;
	AI_RTD_Ch_4_Value 	AT %I* : INT;
	
	//Terminal status
	WcState_WcState AT %I*: BOOL;
	InfoData_State AT %I*: UINT;
	
	//FB-s
	EL3214_Error : FB_TerminalError;
END_VAR

(*
* TODO:
* Status words of the channels
*)

EnO := En;

//Error FB instance
EL3214_Error(
	En := TRUE,
	iTerminal_ID := iTerminal_ID,
	bWcState := WcState_WcState,
	uiInfoData_State := InfoData_State,
	pErrorSystem := ErrorSystem,
	bError => bError,
);

IF En THEN
	IF bError = FALSE THEN
		iAi_Ch1_Value := AI_RTD_Ch_1_Value;
		iAi_Ch2_Value := AI_RTD_Ch_2_Value;
		iAi_Ch3_Value := AI_RTD_Ch_3_Value;
		iAi_Ch4_Value := AI_RTD_Ch_4_Value;
	ELSE
		iAi_Ch1_Value := 0;
		iAi_Ch2_Value := 0;
		iAi_Ch3_Value := 0;
		iAi_Ch4_Value := 0;
	END_IF
END_IF

END_FUNCTION_BLOCK

// tc_mca_std_lib/POUs/Hardware/EtherCAT_Terminals/Analog_Inputs/EL3255
//EL3255 | 5-channel potentiometer measurement with sensor supply
FUNCTION_BLOCK EL3255

VAR_INPUT
	En: BOOL;
	iTerminal_ID : INT;
	ErrorSystem : POINTER TO ST_ErrorSystem;
END_VAR

VAR_OUTPUT
	EnO : BOOL;	
	Ch1_Value : INT;
	Ch2_Value : INT;
	Ch3_Value : INT;
	Ch4_Value : INT;
	Ch5_Value : INT;
	bError : BOOL;
END_VAR

VAR
	AI_Std_Ch1_Value AT %I* : INT;
	AI_Std_Ch2_Value AT %I* : INT;
	AI_Std_Ch3_Value AT %I* : INT;
	AI_Std_Ch4_Value AT %I* : INT;
	AI_Std_Ch5_Value AT %I* : INT;
	WcState_WcState AT %I*: BOOL;
	InfoData_State AT %I*: UINT;
	
	//FB-s
	EL3255_Error : FB_TerminalError;
END_VAR

(*
* TODO:
* Channel Status words
*)

EnO:=En;

//Error FB instance
EL3255_Error(
	En := TRUE,
	iTerminal_ID := iTerminal_ID,
	bWcState := WcState_WcState,
	uiInfoData_State := InfoData_State,
	pErrorSystem := ErrorSystem,
	bError => bError,
);

IF EN THEN
	IF NOT bError THEN
		Ch1_Value := AI_Std_Ch1_Value;
		Ch2_Value := AI_Std_Ch2_Value;
		Ch3_Value := AI_Std_Ch3_Value;
		Ch4_Value := AI_Std_Ch4_Value;
		Ch5_Value := AI_Std_Ch5_Value;
	ELSE
		Ch1_Value := 0;
		Ch2_Value := 0;
		Ch3_Value := 0;
		Ch4_Value := 0;
		Ch5_Value := 0;
	END_IF
END_IF

END_FUNCTION_BLOCK

// tc_mca_std_lib/POUs/Hardware/EtherCAT_Terminals/Analog_Inputs/FB_CalculateFrequency_3702_v0_01
FUNCTION_BLOCK FB_CalculateFrequency_3702_v0_01
VAR CONSTANT
	///200 samples/period
	cBufferSize: INT := 1000;
END_VAR
VAR_INPUT
	En: BOOL;
	bCalculate: BOOL;
	aBufferValue: ARRAY[0..(cBuffersize - 1)] OF INT;
	aBufferDcTime: ARRAY[0..(cBuffersize - 1)] OF UDINT;
	///If curve has a DC offset
	nDCOffset: INT := 0;
END_VAR
VAR_OUTPUT
	EnO: BOOL;
	bError: BOOL;
	fActFrequency: LREAL;
END_VAR
VAR
	nIndex: INT;
	nFirstZeroCrossing: INT;
	nLastZeroCrossing: INT;
	rTimeFirst: REAL := 0;
	rTimeLast: REAL := 0;
	rTimeRes: REAL := 0;
	nCrossings: INT := 0;
END_VAR
VAR_TEMP
	rRange: REAL := 0;
	rTimeSpan: REAL := 0;
END_VAR

EnO:=En;
bError:=FALSE;
nCrossings:=0;
IF En AND bCalculate THEN
	//Serach for crossings of nDCOffset
	FOR nIndex:=1 TO cBuffersize-1 DO
		IF((aBufferValue[nIndex]>nDCOffset AND aBufferValue[nIndex-1]<=nDCOffset) OR (aBufferValue[nIndex]<nDCOffset AND aBufferValue[nIndex-1]>=nDCOffset))	THEN
			IF(nCrossings=0) THEN
				nFirstZeroCrossing:=nIndex;
			END_IF
			nLastZeroCrossing:=nIndex;
			nCrossings:=nCrossings+1;
		END_IF
	END_FOR	
	
	IF nFirstZeroCrossing < nLastZeroCrossing  AND  nCrossings>2 THEN
		//interpolate zero crossings for higher accuracy
		rTimeRes:=UDINT_TO_REAL(aBufferDcTime[1]-aBufferDcTime[0]); //Buffer must contain more than 2 values
		rRange:=INT_TO_REAL(ABS(aBufferValue[nFirstZeroCrossing-1]-aBufferValue[nFirstZeroCrossing]));
		rTimeFirst:=UDINT_TO_REAL( aBufferDcTime[nFirstZeroCrossing-1])+ABS(INT_TO_REAL(aBufferValue[nFirstZeroCrossing-1])/rRange*rTimeRes);
		rRange:=INT_TO_REAL(ABS(aBufferValue[nLastZeroCrossing-1]-aBufferValue[nLastZeroCrossing]));
		rTimeLast:=UDINT_TO_REAL( aBufferDcTime[nLastZeroCrossing-1])+ABS(INT_TO_REAL(aBufferValue[nLastZeroCrossing-1])/rRange*rTimeRes);

		//Time span first to last (considering that max one time counter overflow have occured in the total time range of the time buffer)	
		IF rTimeFirst<rTimeLast THEN		
			rTimeSpan:=rTimeLast-rTimeFirst;
		ELSE //overflow of counter once (only 32bit timestamp =4.29seconds)
			rTimeSpan:=4294967296.0-rTimeFirst+rTimeLast;
		END_IF
		
		fActFrequency:=1000000000.0/rTimeSpan*(nCrossings-1)/2; //two crossings per period => Average frequency over buffer.
	ELSE
		fActFrequency:=0;
	END_IF
END_IF

END_FUNCTION_BLOCK

// tc_mca_std_lib/POUs/Hardware/EtherCAT_Terminals/Digital_Inputs/EL1008
///EL1008 | 8-channel digital input terminal 24 V DC, 3 ms
FUNCTION_BLOCK EL1008

VAR_INPUT
	En: BOOL;
	iTerminal_ID : INT;
	ErrorSystem : POINTER TO ST_ErrorSystem;
END_VAR

VAR_OUTPUT
	EnO: BOOL;
	bDi_1: BOOL;
	bDi_2: BOOL;
	bDi_3: BOOL;
	bDi_4: BOOL;
	bDi_5: BOOL;
	bDi_6: BOOL;
	bDi_7: BOOL;
	bDi_8: BOOL;
	bError: BOOL;
END_VAR

VAR
	Channel_1_Input AT %I*: BOOL;
	Channel_2_Input AT %I*: BOOL;
	Channel_3_Input AT %I*: BOOL;
	Channel_4_Input AT %I*: BOOL;
	Channel_5_Input AT %I*: BOOL;
	Channel_6_Input AT %I*: BOOL;
	Channel_7_Input AT %I*: BOOL;
	Channel_8_Input AT %I*: BOOL;
	WcState_WcState AT %I*: BOOL;
	InfoData_State AT %I*: UINT;
	
	//FB-s
	EL1008_Error : FB_TerminalError;
END_VAR

EnO:=En;

//Error FB instance
EL1008_Error(
	En := TRUE,
	iTerminal_ID := iTerminal_ID,
	bWcState := WcState_WcState,
	uiInfoData_State := InfoData_State,
	pErrorSystem := ErrorSystem,
	bError => bError,
);

IF En THEN
	IF bError=FALSE THEN
		bDi_1:=Channel_1_Input;
		bDi_2:=Channel_2_Input;
		bDi_3:=Channel_3_Input;
		bDi_4:=Channel_4_Input;
		bDi_5:=Channel_5_Input;
		bDi_6:=Channel_6_Input;
		bDi_7:=Channel_7_Input;
		bDi_8:=Channel_8_Input;
	ELSE
		bDi_1:=FALSE;
		bDi_2:=FALSE;
		bDi_3:=FALSE;
		bDi_4:=FALSE;
		bDi_5:=FALSE;
		bDi_6:=FALSE;
		bDi_7:=FALSE;
		bDi_8:=FALSE;
	END_IF
END_IF

END_FUNCTION_BLOCK

// tc_mca_std_lib/POUs/Hardware/EtherCAT_Terminals/Digital_Inputs/EL1018
///EL1018 | 8-channel digital input terminal 24 V DC, 10 µs
FUNCTION_BLOCK EL1018

VAR_INPUT
	En: BOOL;
	iTerminal_ID : INT;
	ErrorSystem : POINTER TO ST_ErrorSystem;
END_VAR

VAR_OUTPUT
	EnO: BOOL;
	bDi_1: BOOL;
	bDi_2: BOOL;
	bDi_3: BOOL;
	bDi_4: BOOL;
	bDi_5: BOOL;
	bDi_6: BOOL;
	bDi_7: BOOL;
	bDi_8: BOOL;
	bError : BOOL;
END_VAR

VAR
	Channel_1_Input AT %I*: BOOL;
	Channel_2_Input AT %I*: BOOL;
	Channel_3_Input AT %I*: BOOL;
	Channel_4_Input AT %I*: BOOL;
	Channel_5_Input AT %I*: BOOL;
	Channel_6_Input AT %I*: BOOL;
	Channel_7_Input AT %I*: BOOL;
	Channel_8_Input AT %I*: BOOL;
	WcState_WcState AT %I*: BOOL;
	InfoData_State  AT %I*: UINT;
	
	//FB-s
	EL1018_Error : FB_TerminalError;
END_VAR

EnO:=En;

//Error FB instance
EL1018_Error(
	En := TRUE,
	iTerminal_ID := iTerminal_ID,
	bWcState := WcState_WcState,
	uiInfoData_State := InfoData_State,
	pErrorSystem := ErrorSystem,
	bError => bError,
);

IF En THEN
	IF bError=FALSE THEN
		bDi_1:=Channel_1_Input;
		bDi_2:=Channel_2_Input;
		bDi_3:=Channel_3_Input;
		bDi_4:=Channel_4_Input;
		bDi_5:=Channel_5_Input;
		bDi_6:=Channel_6_Input;
		bDi_7:=Channel_7_Input;
		bDi_8:=Channel_8_Input;
	ELSE
		bDi_1:=FALSE;
		bDi_2:=FALSE;
		bDi_3:=FALSE;
		bDi_4:=FALSE;
		bDi_5:=FALSE;
		bDi_6:=FALSE;
		bDi_7:=FALSE;
		bDi_8:=FALSE;
	END_IF
END_IF

END_FUNCTION_BLOCK

// tc_mca_std_lib/POUs/Hardware/EtherCAT_Terminals/Digital_Inputs/EL1808
///EL1808 | HD EtherCAT Terminals, 8-channel digital input 24 V DC, 3 ms, 2-wire connection
FUNCTION_BLOCK EL1808

VAR_INPUT
	En: BOOL;
	iTerminal_ID : INT;
	ErrorSystem : POINTER TO ST_ErrorSystem;
END_VAR

VAR_OUTPUT
	EnO: BOOL;
	bDi_1: BOOL;
	bDi_2: BOOL;
	bDi_3: BOOL;
	bDi_4: BOOL;
	bDi_5: BOOL;
	bDi_6: BOOL;
	bDi_7: BOOL;
	bDi_8: BOOL;
	bError: BOOL;
END_VAR

VAR
	Channel_1_Input AT %I*: BOOL;
	Channel_2_Input AT %I*: BOOL;
	Channel_3_Input AT %I*: BOOL;
	Channel_4_Input AT %I*: BOOL;
	Channel_5_Input AT %I*: BOOL;
	Channel_6_Input AT %I*: BOOL;
	Channel_7_Input AT %I*: BOOL;
	Channel_8_Input AT %I*: BOOL;
	WcState_WcState AT %I*: BOOL;
	InfoData_State AT %I*: UINT;
	
	//FB-s
	EL1808_Error : FB_TerminalError;
END_VAR

EnO:=En;

//Error FB instance
EL1808_Error(
	En := TRUE,
	iTerminal_ID := iTerminal_ID,
	bWcState := WcState_WcState,
	uiInfoData_State := InfoData_State,
	pErrorSystem := ErrorSystem,
	bError => bError,
);

IF En THEN
	IF bError=FALSE THEN
		bDi_1:=Channel_1_Input;
		bDi_2:=Channel_2_Input;
		bDi_3:=Channel_3_Input;
		bDi_4:=Channel_4_Input;
		bDi_5:=Channel_5_Input;
		bDi_6:=Channel_6_Input;
		bDi_7:=Channel_7_Input;
		bDi_8:=Channel_8_Input;
	ELSE
		bDi_1:=FALSE;
		bDi_2:=FALSE;
		bDi_3:=FALSE;
		bDi_4:=FALSE;
		bDi_5:=FALSE;
		bDi_6:=FALSE;
		bDi_7:=FALSE;
		bDi_8:=FALSE;
	END_IF
END_IF

END_FUNCTION_BLOCK

// tc_mca_std_lib/POUs/Hardware/EtherCAT_Terminals/Digital_Inputs/EL1809
///EL1809 | HD EtherCAT Terminals, 16-channel digital input 24 V DC, 3 ms
FUNCTION_BLOCK EL1809

VAR_INPUT
	En: BOOL;
	iTerminal_ID : INT;
	ErrorSystem : POINTER TO ST_ErrorSystem;
END_VAR

VAR_OUTPUT
	EnO: BOOL;
	bDi_1: BOOL;
	bDi_2: BOOL;
	bDi_3: BOOL;
	bDi_4: BOOL;
	bDi_5: BOOL;
	bDi_6: BOOL;
	bDi_7: BOOL;
	bDi_8: BOOL;
	bDi_9: BOOL;
	bDi_10: BOOL;
	bDi_11: BOOL;
	bDi_12: BOOL;
	bDi_13: BOOL;
	bDi_14: BOOL;
	bDi_15: BOOL;
	bDi_16: BOOL;
	bError: BOOL;
END_VAR

VAR
	Channel_1_Input AT %I*: BOOL;
	Channel_2_Input AT %I*: BOOL;
	Channel_3_Input AT %I*: BOOL;
	Channel_4_Input AT %I*: BOOL;
	Channel_5_Input AT %I*: BOOL;
	Channel_6_Input AT %I*: BOOL;
	Channel_7_Input AT %I*: BOOL;
	Channel_8_Input AT %I*: BOOL;
	Channel_9_Input AT %I*: BOOL;
	Channel_10_Input AT %I*: BOOL;
	Channel_11_Input AT %I*: BOOL;
	Channel_12_Input AT %I*: BOOL;
	Channel_13_Input AT %I*: BOOL;
	Channel_14_Input AT %I*: BOOL;
	Channel_15_Input AT %I*: BOOL;
	Channel_16_Input AT %I*: BOOL;
	WcState_WcState AT %I*: BOOL;
	InfoData_State AT %I*: UINT;
	
	//FB-s
	EL1809_Error : FB_TerminalError;
END_VAR

EnO:=En;

//Error FB instance
EL1809_Error(
	En := TRUE,
	iTerminal_ID := iTerminal_ID,
	bWcState := WcState_WcState,
	uiInfoData_State := InfoData_State,
	pErrorSystem := ErrorSystem,
	bError => bError,
);

IF En THEN
	IF bError=FALSE THEN
		bDi_1:=Channel_1_Input;
		bDi_2:=Channel_2_Input;
		bDi_3:=Channel_3_Input;
		bDi_4:=Channel_4_Input;
		bDi_5:=Channel_5_Input;
		bDi_6:=Channel_6_Input;
		bDi_7:=Channel_7_Input;
		bDi_8:=Channel_8_Input;
		bDi_9:=Channel_9_Input;
		bDi_10:=Channel_10_Input;
		bDi_11:=Channel_11_Input;
		bDi_12:=Channel_12_Input;
		bDi_13:=Channel_13_Input;
		bDi_14:=Channel_14_Input;
		bDi_15:=Channel_15_Input;
		bDi_16:=Channel_16_Input;
	ELSE
		bDi_1:=FALSE;
		bDi_2:=FALSE;
		bDi_3:=FALSE;
		bDi_4:=FALSE;
		bDi_5:=FALSE;
		bDi_6:=FALSE;
		bDi_7:=FALSE;
		bDi_8:=FALSE;
		bDi_9:=FALSE;
		bDi_10:=FALSE;
		bDi_11:=FALSE;
		bDi_12:=FALSE;
		bDi_13:=FALSE;
		bDi_14:=FALSE;
		bDi_15:=FALSE;
		bDi_16:=FALSE;
	END_IF
END_IF

END_FUNCTION_BLOCK

// tc_mca_std_lib/POUs/Hardware/EtherCAT_Terminals/Digital_Inputs/EL1819
///EL1819 | HD EtherCAT Terminals, 16-channel digital input 24 V DC, 10 µs
FUNCTION_BLOCK EL1819

VAR_INPUT
	En: BOOL;
	iTerminal_ID : INT;
	ErrorSystem : POINTER TO ST_ErrorSystem;
END_VAR

VAR_OUTPUT
	EnO: BOOL;
	bDi_1: BOOL;
	bDi_2: BOOL;
	bDi_3: BOOL;
	bDi_4: BOOL;
	bDi_5: BOOL;
	bDi_6: BOOL;
	bDi_7: BOOL;
	bDi_8: BOOL;
	bDi_9: BOOL;
	bDi_10: BOOL;
	bDi_11: BOOL;
	bDi_12: BOOL;
	bDi_13: BOOL;
	bDi_14: BOOL;
	bDi_15: BOOL;
	bDi_16: BOOL;
	bError: BOOL;
END_VAR

VAR
	Channel_1_Input AT %I*: BOOL;
	Channel_2_Input AT %I*: BOOL;
	Channel_3_Input AT %I*: BOOL;
	Channel_4_Input AT %I*: BOOL;
	Channel_5_Input AT %I*: BOOL;
	Channel_6_Input AT %I*: BOOL;
	Channel_7_Input AT %I*: BOOL;
	Channel_8_Input AT %I*: BOOL;
	Channel_9_Input AT %I*: BOOL;
	Channel_10_Input AT %I*: BOOL;
	Channel_11_Input AT %I*: BOOL;
	Channel_12_Input AT %I*: BOOL;
	Channel_13_Input AT %I*: BOOL;
	Channel_14_Input AT %I*: BOOL;
	Channel_15_Input AT %I*: BOOL;
	Channel_16_Input AT %I*: BOOL;
	WcState_WcState AT %I*: BOOL;
	InfoData_State AT %I*: UINT;
	
	//FB-s
	EL1819_Error : FB_TerminalError;
END_VAR

EnO:=En;

//Error FB instance
EL1819_Error(
	En := TRUE,
	iTerminal_ID := iTerminal_ID,
	bWcState := WcState_WcState,
	uiInfoData_State := InfoData_State,
	pErrorSystem := ErrorSystem,
	bError => bError,
);

IF En THEN
	IF bError=FALSE THEN
		bDi_1:=Channel_1_Input;
		bDi_2:=Channel_2_Input;
		bDi_3:=Channel_3_Input;
		bDi_4:=Channel_4_Input;
		bDi_5:=Channel_5_Input;
		bDi_6:=Channel_6_Input;
		bDi_7:=Channel_7_Input;
		bDi_8:=Channel_8_Input;
		bDi_9:=Channel_9_Input;
		bDi_10:=Channel_10_Input;
		bDi_11:=Channel_11_Input;
		bDi_12:=Channel_12_Input;
		bDi_13:=Channel_13_Input;
		bDi_14:=Channel_14_Input;
		bDi_15:=Channel_15_Input;
		bDi_16:=Channel_16_Input;
	ELSE
		bDi_1:=FALSE;
		bDi_2:=FALSE;
		bDi_3:=FALSE;
		bDi_4:=FALSE;
		bDi_5:=FALSE;
		bDi_6:=FALSE;
		bDi_7:=FALSE;
		bDi_8:=FALSE;
		bDi_9:=FALSE;
		bDi_10:=FALSE;
		bDi_11:=FALSE;
		bDi_12:=FALSE;
		bDi_13:=FALSE;
		bDi_14:=FALSE;
		bDi_15:=FALSE;
		bDi_16:=FALSE;
	END_IF
END_IF

END_FUNCTION_BLOCK

// tc_mca_std_lib/POUs/Hardware/EtherCAT_Terminals/Digital_Inputs/FB_EL1252ASM_v1_00
FUNCTION_BLOCK FB_EL1252ASM_v1_00
VAR_INPUT
	En: BOOL;
END_VAR
VAR_OUTPUT
	EnO: BOOL;
	Di_1: BOOL;
	Di_2: BOOL;
	Di_1_LatchTimePos: ULINT;
	Di_2_LatchTimePos: ULINT;
	Di_1_LatchTimeNeg: ULINT;
	Di_2_LatchTimeNeg: ULINT;
	///Below bits can be used but then they must be enabled in the COE of the card. Nicklas suggested to not use these (since something wss written that you then only were allowed to read the latch time onece (some kkind of auto reset??))	
	///Di_1_LatchNeg:BOOL;
	///	Di_1_LatchPos:BOOL;
	///	Di_2_LatchNeg:BOOL;
	///	Di_2_LatchPos:BOOL;
	Error: BOOL;
END_VAR
VAR
	Channel_1_Input AT %I*: BOOL;
	Channel_2_Input AT %I*: BOOL;
	///Latch_Status1 AT %I*: USINT;
	///	Latch_Status2 AT %I*: USINT;
	Latch_LatchPos1 AT %I*: ULINT;
	Latch_LatchNeg1 AT %I*: ULINT;
	Latch_LatchPos2 AT %I*: ULINT;
	Latch_LatchNeg2 AT %I*: ULINT;
	WcState_WcState AT %I*: BOOL;
	InfoData_State AT %I*: UINT;
END_VAR

EnO:=En;

IF En AND (WcState_WcState OR InfoData_State<>16#8) THEN //InfoData_State==0 => in OP mode
	Error:=TRUE;
ELSE
	Error:=FALSE;
END_IF

IF En THEN
	IF Error=FALSE THEN
		Di_1:=Channel_1_Input;
		Di_2:=Channel_2_Input;
	(*	Di_1_LatchPos:=Latch_Status1.0;
		Di_1_LatchNeg:=Latch_Status1.1;
		Di_2_LatchPos:=Latch_Status2.0;
		Di_2_LatchNeg:=Latch_Status2.1;*)
		Di_1_LatchTimePos:=Latch_LatchPos1;
		Di_2_LatchTimePos:=Latch_LatchPos2;		
		Di_1_LatchTimeNeg:=Latch_LatchNeg1;		
		Di_2_LatchTimeNeg:=Latch_LatchNeg2;
		
	ELSE
		Di_1:=FALSE;
		Di_2:=FALSE;
	END_IF
END_IF

END_FUNCTION_BLOCK

// tc_mca_std_lib/POUs/Hardware/EtherCAT_Terminals/Digital_Outputs/EL2014
FUNCTION_BLOCK EL2014
VAR_INPUT
	En: BOOL;
	iTerminal_ID : INT; 
	bDo_1: BOOL;
	bDo_2: BOOL;
	bDo_3: BOOL;
	bDo_4: BOOL;
	ErrorSystem : POINTER TO ST_ErrorSystem;
END_VAR

VAR_OUTPUT
	EnO : BOOL;
	bError : BOOL;
END_VAR

VAR
	Channel_1_Output AT %Q*: BOOL;
	Channel_2_Output AT %Q*: BOOL;
	Channel_3_Output AT %Q*: BOOL;
	Channel_4_Output AT %Q*: BOOL;
	WcState_WcState AT %I*: BOOL;
	InfoData_State AT %I*: UINT;
	
	//FB-s
	EL2014_Error : FB_TerminalError;
END_VAR

(*
* TODO:
* Channel diagnostic variables and device diag variables
*)

EnO:=En;

EL2014_Error(
	En := TRUE,
	iTerminal_ID := iTerminal_ID,
	bWcState := WcState_WcState,
	uiInfoData_State := InfoData_State,
	pErrorSystem := ErrorSystem,
	bError => bError,
);

IF En THEN
	IF bError=FALSE THEN
		Channel_1_Output:=bDo_1;
		Channel_2_Output:=bDo_2;
		Channel_3_Output:=bDo_3;
		Channel_4_Output:=bDo_4;
	ELSE
		Channel_1_Output:=FALSE;
		Channel_2_Output:=FALSE;
		Channel_3_Output:=FALSE;
		Channel_4_Output:=FALSE;
	END_IF
END_IF

END_FUNCTION_BLOCK

// tc_mca_std_lib/POUs/Hardware/EtherCAT_Terminals/Digital_Outputs/EL2252
///EL2252 | XFC, 2-channel digital output terminal with time stamp, tri-state
FUNCTION_BLOCK EL2252
VAR_INPUT
	En: BOOL;
	iTerminal_ID : INT; 
	bDo_1: BOOL;
	bDo_2: BOOL;
ErrorSystem : POINTER TO ST_ErrorSystem;
END_VAR

VAR_OUTPUT
	EnO : BOOL;
	bError : BOOL;
END_VAR

VAR
	Channel_1_Output AT %Q*: BOOL;
	Channel_2_Output AT %Q*: BOOL;
	WcState_WcState AT %I*: BOOL;
	InfoData_State AT %I*: UINT;
	
	//FB-s
	EL2252_Error : FB_TerminalError;
END_VAR

(*
* TODO:
* Add the DC sync variables
*)

EL2252_Error(
	En := TRUE,
	iTerminal_ID := iTerminal_ID,
	bWcState := WcState_WcState,
	uiInfoData_State := InfoData_State,
	pErrorSystem := ErrorSystem,
	bError => bError,
);

IF En THEN
	IF bError=FALSE THEN
		Channel_1_Output:=bDo_1;
		Channel_2_Output:=bDo_2;
	ELSE
		Channel_1_Output:=FALSE;
		Channel_2_Output:=FALSE;
	END_IF
END_IF

END_FUNCTION_BLOCK

// tc_mca_std_lib/POUs/Hardware/EtherCAT_Terminals/Digital_Outputs/EL2808
FUNCTION_BLOCK EL2808

VAR_INPUT
	En: BOOL;
	iTerminal_ID : INT; 
	bDo_1: BOOL;
	bDo_2: BOOL;
	bDo_3: BOOL;
	bDo_4: BOOL;
	bDo_5: BOOL;
	bDo_6: BOOL;
	bDo_7: BOOL;
	bDo_8: BOOL;
	ErrorSystem : POINTER TO ST_ErrorSystem;
END_VAR

VAR_OUTPUT
	EnO : BOOL;
	bError : BOOL;
END_VAR

VAR
	Channel_1_Output AT %Q*: BOOL;
	Channel_2_Output AT %Q*: BOOL;
	Channel_3_Output AT %Q*: BOOL;
	Channel_4_Output AT %Q*: BOOL;
	Channel_5_Output AT %Q*: BOOL;
	Channel_6_Output AT %Q*: BOOL;
	Channel_7_Output AT %Q*: BOOL;
	Channel_8_Output AT %Q*: BOOL;
	WcState_WcState AT %I*: BOOL;
	InfoData_State AT %I*: UINT;
	
	//FB-s
	EL2808_Error : FB_TerminalError;
END_VAR

EnO:=En;

EL2808_Error(
	En := TRUE,
	iTerminal_ID := iTerminal_ID,
	bWcState := WcState_WcState,
	uiInfoData_State := InfoData_State,
	pErrorSystem := ErrorSystem,
	bError => bError,
);

IF En THEN
	IF bError=FALSE THEN
		Channel_1_Output:=bDo_1;
		Channel_2_Output:=bDo_2;
		Channel_3_Output:=bDo_3;
		Channel_4_Output:=bDo_4;
		Channel_5_Output:=bDo_5;
		Channel_6_Output:=bDo_6;
		Channel_7_Output:=bDo_7;
		Channel_8_Output:=bDo_8;
	ELSE
		Channel_1_Output:=FALSE;
		Channel_2_Output:=FALSE;
		Channel_3_Output:=FALSE;
		Channel_4_Output:=FALSE;
		Channel_5_Output:=FALSE;
		Channel_6_Output:=FALSE;
		Channel_7_Output:=FALSE;
		Channel_8_Output:=FALSE;
	END_IF
END_IF

END_FUNCTION_BLOCK

// tc_mca_std_lib/POUs/Hardware/EtherCAT_Terminals/Digital_Outputs/EL2819
FUNCTION_BLOCK EL2819
VAR_INPUT
	En: BOOL;
	iTerminal_ID : INT; 
	bDo_1: BOOL;
	bDo_2: BOOL;
	bDo_3: BOOL;
	bDo_4: BOOL;
	bDo_5: BOOL;
	bDo_6: BOOL;
	bDo_7: BOOL;
	bDo_8: BOOL;
	bDo_9: BOOL;
	bDo_10: BOOL;
	bDo_11: BOOL;
	bDo_12: BOOL;
	bDo_13: BOOL;
	bDo_14: BOOL;
	bDo_15: BOOL;
	bDo_16: BOOL;
	ErrorSystem : POINTER TO ST_ErrorSystem;
END_VAR

VAR_OUTPUT
	EnO : BOOL;
	bError : BOOL;
END_VAR

VAR
	Channel_1_Output AT %Q*: BOOL;
	Channel_2_Output AT %Q*: BOOL;
	Channel_3_Output AT %Q*: BOOL;
	Channel_4_Output AT %Q*: BOOL;
	Channel_5_Output AT %Q*: BOOL;
	Channel_6_Output AT %Q*: BOOL;
	Channel_7_Output AT %Q*: BOOL;
	Channel_8_Output AT %Q*: BOOL;
	Channel_9_Output AT %Q*: BOOL;
	Channel_10_Output AT %Q*: BOOL;
	Channel_11_Output AT %Q*: BOOL;
	Channel_12_Output AT %Q*: BOOL;
	Channel_13_Output AT %Q*: BOOL;
	Channel_14_Output AT %Q*: BOOL;
	Channel_15_Output AT %Q*: BOOL;
	Channel_16_Output AT %Q*: BOOL;
	
	WcState_WcState AT %I*: BOOL;
	InfoData_State AT %I*: UINT;
	
	//FB-s
	EL2819_Error : FB_TerminalError;
END_VAR

(*
* TODO:
* Channel diagnostic variables and device diag variables
*)

EnO:=En;

EL2819_Error(
	En := TRUE,
	iTerminal_ID := iTerminal_ID,
	bWcState := WcState_WcState,
	uiInfoData_State := InfoData_State,
	pErrorSystem := ErrorSystem,
	bError => bError,
);

IF En THEN
	IF bError=FALSE THEN
		Channel_1_Output:=bDo_1;
		Channel_2_Output:=bDo_2;
		Channel_3_Output:=bDo_3;
		Channel_4_Output:=bDo_4;
		Channel_5_Output:=bDo_5;
		Channel_6_Output:=bDo_6;
		Channel_7_Output:=bDo_7;
		Channel_8_Output:=bDo_8;
		Channel_9_Output:=bDo_9;
		Channel_10_Output:=bDo_10;
		Channel_11_Output:=bDo_11;
		Channel_12_Output:=bDo_12;
		Channel_13_Output:=bDo_13;
		Channel_14_Output:=bDo_14;
		Channel_15_Output:=bDo_15;
		Channel_16_Output:=bDo_16;
	ELSE
		Channel_1_Output:=FALSE;
		Channel_2_Output:=FALSE;
		Channel_3_Output:=FALSE;
		Channel_4_Output:=FALSE;
		Channel_5_Output:=FALSE;
		Channel_6_Output:=FALSE;
		Channel_7_Output:=FALSE;
		Channel_8_Output:=FALSE;
		Channel_9_Output:=FALSE;
		Channel_10_Output:=FALSE;
		Channel_11_Output:=FALSE;
		Channel_12_Output:=FALSE;
		Channel_13_Output:=FALSE;
		Channel_14_Output:=FALSE;
		Channel_15_Output:=FALSE;
		Channel_16_Output:=FALSE;
	END_IF
END_IF

END_FUNCTION_BLOCK

// tc_mca_std_lib/POUs/Hardware/EtherCAT_Terminals/Measuring_Terminals/EL5002
//EL5002 | 2-chennel SSI absolute encoder terminal
FUNCTION_BLOCK EL5002

VAR_INPUT
	En: BOOL;
	iTerminal_ID : INT;
	ErrorSystem : POINTER TO ST_ErrorSystem;
END_VAR

VAR_OUTPUT
	EnO: BOOL;
	Ch1_Counter_Value : UDINT;
	Ch2_Counter_Value : UDINT;
	bError: BOOL;
END_VAR

VAR
	udi_Ch1_Cnt_Value AT %I* : UDINT;
	udi_Ch2_Cnt_Value AT %I* : UDINT;
	WcState_WcState AT %I*: BOOL;
	InfoData_State AT %I*: UINT;
	
	//FB-s
	EL5002_Error : FB_TerminalError;
END_VAR

(*
* TODO:
* Channel Status words
*)

EnO:=En;

//Error FB instance
EL5002_Error(
	En := TRUE,
	iTerminal_ID := iTerminal_ID,
	bWcState := WcState_WcState,
	uiInfoData_State := InfoData_State,
	pErrorSystem := ErrorSystem,
	bError => bError,
);

IF EN THEN
	IF NOT bError THEN
		Ch1_Counter_Value := udi_Ch1_Cnt_Value;
		Ch2_Counter_Value := udi_Ch2_Cnt_Value;
	ELSE
		Ch1_Counter_Value := 0;
		Ch2_Counter_Value := 0;
	END_IF
END_IF

END_FUNCTION_BLOCK

// tc_mca_std_lib/POUs/Hardware/EtherCAT_Terminals/Measuring_Terminals/EL5021
//EL5021 | 1-channel Sin/Cos encoder
FUNCTION_BLOCK EL5021

VAR_INPUT
	En: BOOL;
	iTerminal_ID : INT;
	ErrorSystem : POINTER TO ST_ErrorSystem;
END_VAR

VAR_OUTPUT
	EnO: BOOL;
	Counter_Value : UDINT;
	Latch_Value : UDINT;
	bError: BOOL;
END_VAR

VAR
	udiCounter_Value AT %I* : UDINT;
	udiLatch_Value AT %I* : UDINT;
	WcState_WcState AT %I*: BOOL;
	InfoData_State AT %I*: UINT;
	
	//FB-s
	EL5021_Error : FB_TerminalError;
END_VAR

(*
* TODO:
* Channel Status words, control words
*)

EnO:=En;

//Error FB instance
EL5021_Error(
	En := TRUE,
	iTerminal_ID := iTerminal_ID,
	bWcState := WcState_WcState,
	uiInfoData_State := InfoData_State,
	pErrorSystem := ErrorSystem,
	bError => bError,
);

IF EN THEN
	IF NOT bError THEN
		Counter_Value := udiCounter_Value;
		Latch_Value := udiLatch_Value;
	ELSE
		Counter_Value := 0;
		Latch_Value := 0;
	END_IF
END_IF

END_FUNCTION_BLOCK

// tc_mca_std_lib/POUs/Hardware/EtherCAT_Terminals/Measuring_Terminals/EL5042
//EL5042 | 2-channel BiSS-C absolute encoder terminal
FUNCTION_BLOCK EL5042

VAR_INPUT
	En: BOOL;
	iTerminal_ID : INT;
	ErrorSystem : POINTER TO ST_ErrorSystem;
END_VAR

VAR_OUTPUT
	EnO: BOOL;
	Ch1_Position : ULINT;
	Ch2_Position : ULINT;
	bError: BOOL;
END_VAR

